(* Logix 5000 project; controller VET 1756-L62 rev 19.52; software revision 19.01; part 8 of 27 *)

        [27].Data.tolva[7] := 17, [27].Data.tolva[8] := 18, [27].Data.tolva[9] := 19, [27].Data.tolva[10] := 20, [27].Data.tolva[11] := 29, [27].Data.tolva[12] := 26, [27].Data.tolva[13] := 27, [27].Data.tolva[14] := 28, [27].Data.tolva[15] := 21, [27].Data.tolva[16] := 38, [27].Data.lugar[0] := 1, [27].Data.lugar[1] := 1, [27].Data.lugar[2] := 1, [27].Data.lugar[3] := 1, [27].Data.lugar[4] := 2, [27].Data.lugar[5] := 2, [27].Data.lugar[6] := 2, [27].Data.lugar[7] := 2, [27].Data.lugar[8] := 3, [27].Data.lugar[9] := 3, [27].Data.lugar[10] := 3, [27].Data.lugar[11] := 4, [27].Data.lugar[12] := 4, [27].Data.lugar[13] := 4, [27].Data.lugar[14] := 4, [27].Data.lugar[15] := 3, [27].Data.lugar[16] := 6, [27].Data.flags[0] := 5, [27].Data.flags[1] := 5, [27].Data.flags[2] := 5, [27].Data.flags[3] := 5, [27].Data.flags[4] := 5, [27].Data.flags[5] := 5, [27].Data.flags[6] := 5, [27].Data.flags[7] := 5, [27].Data.flags[8] := 5, [27].Data.flags[9] := 5, [27].Data.flags[10] := 5, [27].Data.flags[11] := 5, [27].Data.flags[12] := 5, [27].Data.flags[13] := 5, [27].Data.flags[14] := 5, [27].Data.flags[15] := 5, [27].Data.flags[16] := 5, [27].Data.fecha_i[0] := 20140324, [27].Data.fecha_i[1] := 20140324, [27].Data.fecha_i[2] := 20140324, [27].Data.fecha_i[3] := 20140324, [27].Data.fecha_i[4] := 20140324, [27].Data.fecha_i[5] := 20140324, [27].Data.fecha_i[6] := 20140324, [27].Data.fecha_i[7] := 20140324, [27].Data.fecha_i[8] := 20140324, [27].Data.fecha_i[9] := 20140324, [27].Data.fecha_i[10] := 20140324, [27].Data.fecha_i[11] := 20140324, [27].Data.fecha_i[12] := 20140324, [27].Data.fecha_i[13] := 20140324, [27].Data.fecha_i[14] := 20140324, [27].Data.fecha_i[15] := 20140324,
        [27].Data.fecha_i[16] := 20140324, [27].Data.fecha_f[0] := 20140324, [27].Data.fecha_f[1] := 20140324, [27].Data.fecha_f[2] := 20140324, [27].Data.fecha_f[3] := 20140324, [27].Data.fecha_f[4] := 20140324, [27].Data.fecha_f[5] := 20140324, [27].Data.fecha_f[6] := 20140324, [27].Data.fecha_f[7] := 20140324, [27].Data.fecha_f[8] := 20140324, [27].Data.fecha_f[9] := 20140324, [27].Data.fecha_f[10] := 20140324, [27].Data.fecha_f[11] := 20140324, [27].Data.fecha_f[12] := 20140324, [27].Data.fecha_f[13] := 20140324, [27].Data.fecha_f[14] := 20140324, [27].Data.fecha_f[15] := 20140324, [27].Data.fecha_f[16] := 20140324, [27].Data.hora_i[0] := 16373539, [27].Data.hora_i[1] := 16375259, [27].Data.hora_i[2] := 16380789, [27].Data.hora_i[3] := 16381714, [27].Data.hora_i[4] := 16373539, [27].Data.hora_i[5] := 16374674, [27].Data.hora_i[6] := 16375794, [27].Data.hora_i[7] := 16380539, [27].Data.hora_i[8] := 16373539, [27].Data.hora_i[9] := 16383864, [27].Data.hora_i[10] := 16393569, [27].Data.hora_i[11] := 16373539, [27].Data.hora_i[12] := 16381754, [27].Data.hora_i[13] := 16392074, [27].Data.hora_i[14] := 16393769, [27].Data.hora_i[15] := 16401384, [27].Data.hora_i[16] := 16404659, [27].Data.hora_f[0] := 16375239, [27].Data.hora_f[1] := 16380769, [27].Data.hora_f[2] := 16381694, [27].Data.hora_f[3] := 16382799, [27].Data.hora_f[4] := 16374654, [27].Data.hora_f[5] := 16375774, [27].Data.hora_f[6] := 16380519, [27].Data.hora_f[7] := 16381269, [27].Data.hora_f[8] := 16383844, [27].Data.hora_f[9] := 16393549, [27].Data.hora_f[10] := 16401364, [27].Data.hora_f[11] := 16381734, [27].Data.hora_f[12] := 16392054, [27].Data.hora_f[13] := 16393749, [27].Data.hora_f[14] := 16394869, [27].Data.hora_f[15] := 16402879, [27].Data.hora_f[16] := 16412864, [28].Head.folio := 40, [28].Head.orden := -3, [28].Head.formula := 'DUMMY$00$00$00$00$00', [28].Head.correlativo := 20, [28].Head.total_batch := 20, [28].Head.peso_teorico := 1733.0, [28].Data.codigo[0] := 51, [28].Data.codigo[1] := 53,
        [28].Data.codigo[2] := 55, [28].Data.codigo[3] := 57, [28].Data.codigo[4] := 60, [28].Data.codigo[5] := 62, [28].Data.codigo[6] := 64, [28].Data.codigo[7] := 66, [28].Data.codigo[8] := 67, [28].Data.codigo[9] := 68, [28].Data.codigo[10] := 69, [28].Data.codigo[11] := 70, [28].Data.codigo[12] := 74, [28].Data.codigo[13] := 75, [28].Data.codigo[14] := 76, [28].Data.codigo[15] := 77, [28].Data.codigo[16] := 81, [28].Data.peso_f[0] := 400.0, [28].Data.peso_f[1] := 350.0, [28].Data.peso_f[2] := 175.0, [28].Data.peso_f[3] := 225.0, [28].Data.peso_f[4] := 125.0, [28].Data.peso_f[5] := 125.0, [28].Data.peso_f[6] := 65.0, [28].Data.peso_f[7] := 65.0, [28].Data.peso_f[8] := 30.0, [28].Data.peso_f[9] := 25.0, [28].Data.peso_f[10] := 17.5, [28].Data.peso_f[11] := 17.5, [28].Data.peso_f[12] := 30.0, [28].Data.peso_f[13] := 5.0, [28].Data.peso_f[14] := 4.0, [28].Data.peso_f[15] := 4.0, [28].Data.peso_f[16] := 70.0, [28].Data.peso_r[0] := 400.74557, [28].Data.peso_r[1] := 350.39438, [28].Data.peso_r[2] := 175.42383, [28].Data.peso_r[3] := 225.02985, [28].Data.peso_r[4] := 125.35709, [28].Data.peso_r[5] := 125.35757, [28].Data.peso_r[6] := 64.76077, [28].Data.peso_r[7] := 65.17856, [28].Data.peso_r[8] := 29.994562, [28].Data.peso_r[9] := 25.012438, [28].Data.peso_r[10] := 17.509579, [28].Data.peso_r[11] := 17.489931, [28].Data.peso_r[12] := 30.008417, [28].Data.peso_r[13] := 5.02573, [28].Data.peso_r[14] := 3.9976578, [28].Data.peso_r[15] := 4.004547, [28].Data.peso_r[16] := 70.10179, [28].Data.tolva[0] := 2, [28].Data.tolva[1] := 4, [28].Data.tolva[2] := 10, [28].Data.tolva[3] := 12, [28].Data.tolva[4] := 7, [28].Data.tolva[5] := 9, [28].Data.tolva[6] := 15, [28].Data.tolva[7] := 17, [28].Data.tolva[8] := 18, [28].Data.tolva[9] := 19, [28].Data.tolva[10] := 20,
        [28].Data.tolva[11] := 29, [28].Data.tolva[12] := 26, [28].Data.tolva[13] := 27, [28].Data.tolva[14] := 28, [28].Data.tolva[15] := 21, [28].Data.tolva[16] := 38, [28].Data.lugar[0] := 1, [28].Data.lugar[1] := 1, [28].Data.lugar[2] := 1, [28].Data.lugar[3] := 1, [28].Data.lugar[4] := 2, [28].Data.lugar[5] := 2, [28].Data.lugar[6] := 2, [28].Data.lugar[7] := 2, [28].Data.lugar[8] := 3, [28].Data.lugar[9] := 3, [28].Data.lugar[10] := 3, [28].Data.lugar[11] := 4, [28].Data.lugar[12] := 4, [28].Data.lugar[13] := 4, [28].Data.lugar[14] := 4, [28].Data.lugar[15] := 3, [28].Data.lugar[16] := 6, [28].Data.flags[0] := 5, [28].Data.flags[1] := 5, [28].Data.flags[2] := 5, [28].Data.flags[3] := 5, [28].Data.flags[4] := 5, [28].Data.flags[5] := 5, [28].Data.flags[6] := 5, [28].Data.flags[7] := 5, [28].Data.flags[8] := 5, [28].Data.flags[9] := 5, [28].Data.flags[10] := 5, [28].Data.flags[11] := 5, [28].Data.flags[12] := 5, [28].Data.flags[13] := 5, [28].Data.flags[14] := 5, [28].Data.flags[15] := 5, [28].Data.flags[16] := 5, [28].Data.fecha_i[0] := 20140324, [28].Data.fecha_i[1] := 20140324, [28].Data.fecha_i[2] := 20140324, [28].Data.fecha_i[3] := 20140324, [28].Data.fecha_i[4] := 20140324, [28].Data.fecha_i[5] := 20140324, [28].Data.fecha_i[6] := 20140324, [28].Data.fecha_i[7] := 20140324, [28].Data.fecha_i[8] := 20140324, [28].Data.fecha_i[9] := 20140324, [28].Data.fecha_i[10] := 20140324, [28].Data.fecha_i[11] := 20140324, [28].Data.fecha_i[12] := 20140324, [28].Data.fecha_i[13] := 20140324, [28].Data.fecha_i[14] := 20140324, [28].Data.fecha_i[15] := 20140324, [28].Data.fecha_i[16] := 20140324, [28].Data.fecha_f[0] := 20140324, [28].Data.fecha_f[1] := 20140324, [28].Data.fecha_f[2] := 20140324,
        [28].Data.fecha_f[3] := 20140324, [28].Data.fecha_f[4] := 20140324, [28].Data.fecha_f[5] := 20140324, [28].Data.fecha_f[6] := 20140324, [28].Data.fecha_f[7] := 20140324, [28].Data.fecha_f[8] := 20140324, [28].Data.fecha_f[9] := 20140324, [28].Data.fecha_f[10] := 20140324, [28].Data.fecha_f[11] := 20140324, [28].Data.fecha_f[12] := 20140324, [28].Data.fecha_f[13] := 20140324, [28].Data.fecha_f[14] := 20140324, [28].Data.fecha_f[15] := 20140324, [28].Data.fecha_f[16] := 20140324, [28].Data.hora_i[0] := 16404664, [28].Data.hora_i[1] := 16410379, [28].Data.hora_i[2] := 16411914, [28].Data.hora_i[3] := 16412839, [28].Data.hora_i[4] := 16404664, [28].Data.hora_i[5] := 16405794, [28].Data.hora_i[6] := 16410919, [28].Data.hora_i[7] := 16411659, [28].Data.hora_i[8] := 16404664, [28].Data.hora_i[9] := 16414989, [28].Data.hora_i[10] := 16424699, [28].Data.hora_i[11] := 16404664, [28].Data.hora_i[12] := 16412859, [28].Data.hora_i[13] := 16423174, [28].Data.hora_i[14] := 16424899, [28].Data.hora_i[15] := 16432524, [28].Data.hora_i[16] := 16435814, [28].Data.hora_f[0] := 16410359, [28].Data.hora_f[1] := 16411894, [28].Data.hora_f[2] := 16412819, [28].Data.hora_f[3] := 16413919, [28].Data.hora_f[4] := 16405774, [28].Data.hora_f[5] := 16410899, [28].Data.hora_f[6] := 16411639, [28].Data.hora_f[7] := 16412374, [28].Data.hora_f[8] := 16414969, [28].Data.hora_f[9] := 16424679, [28].Data.hora_f[10] := 16432504, [28].Data.hora_f[11] := 16412839, [28].Data.hora_f[12] := 16423154, [28].Data.hora_f[13] := 16424879, [28].Data.hora_f[14] := 16425994, [28].Data.hora_f[15] := 16434029, [28].Data.hora_f[16] := 16444014, [29].Head.folio := 40, [29].Head.orden := -3, [29].Head.formula := 'DUMMY$00$00$00$00$00', [29].Head.correlativo := 20, [29].Head.total_batch := 20, [29].Head.peso_teorico := 1733.0, [29].Data.codigo[0] := 51, [29].Data.codigo[1] := 53, [29].Data.codigo[2] := 55, [29].Data.codigo[3] := 57, [29].Data.codigo[4] := 60, [29].Data.codigo[5] := 62,
        [29].Data.codigo[6] := 64, [29].Data.codigo[7] := 66, [29].Data.codigo[8] := 67, [29].Data.codigo[9] := 68, [29].Data.codigo[10] := 69, [29].Data.codigo[11] := 70, [29].Data.codigo[12] := 74, [29].Data.codigo[13] := 75, [29].Data.codigo[14] := 76, [29].Data.codigo[15] := 77, [29].Data.codigo[16] := 81, [29].Data.peso_f[0] := 400.0, [29].Data.peso_f[1] := 350.0, [29].Data.peso_f[2] := 175.0, [29].Data.peso_f[3] := 225.0, [29].Data.peso_f[4] := 125.0, [29].Data.peso_f[5] := 125.0, [29].Data.peso_f[6] := 65.0, [29].Data.peso_f[7] := 65.0, [29].Data.peso_f[8] := 30.0, [29].Data.peso_f[9] := 25.0, [29].Data.peso_f[10] := 17.5, [29].Data.peso_f[11] := 17.5, [29].Data.peso_f[12] := 30.0, [29].Data.peso_f[13] := 5.0, [29].Data.peso_f[14] := 4.0, [29].Data.peso_f[15] := 4.0, [29].Data.peso_f[16] := 70.0, [29].Data.peso_r[0] := 399.58698, [29].Data.peso_r[1] := 350.3239, [29].Data.peso_r[2] := 175.83856, [29].Data.peso_r[3] := 224.96136, [29].Data.peso_r[4] := 124.67243, [29].Data.peso_r[5] := 125.35696, [29].Data.peso_r[6] := 65.3768, [29].Data.peso_r[7] := 64.766815, [29].Data.peso_r[8] := 29.994562, [29].Data.peso_r[9] := 25.012411, [29].Data.peso_r[10] := 17.509384, [29].Data.peso_r[11] := 17.509584, [29].Data.peso_r[12] := 29.994238, [29].Data.peso_r[13] := 4.9850006, [29].Data.peso_r[14] := 4.00441, [29].Data.peso_r[15] := 4.002121, [29].Data.peso_r[16] := 70.10178, [29].Data.tolva[0] := 2, [29].Data.tolva[1] := 4, [29].Data.tolva[2] := 10, [29].Data.tolva[3] := 12, [29].Data.tolva[4] := 7, [29].Data.tolva[5] := 9, [29].Data.tolva[6] := 15, [29].Data.tolva[7] := 17, [29].Data.tolva[8] := 18, [29].Data.tolva[9] := 19, [29].Data.tolva[10] := 20, [29].Data.tolva[11] := 29, [29].Data.tolva[12] := 26, [29].Data.tolva[13] := 27, [29].Data.tolva[14] := 28,
        [29].Data.tolva[15] := 21, [29].Data.tolva[16] := 38, [29].Data.lugar[0] := 1, [29].Data.lugar[1] := 1, [29].Data.lugar[2] := 1, [29].Data.lugar[3] := 1, [29].Data.lugar[4] := 2, [29].Data.lugar[5] := 2, [29].Data.lugar[6] := 2, [29].Data.lugar[7] := 2, [29].Data.lugar[8] := 3, [29].Data.lugar[9] := 3, [29].Data.lugar[10] := 3, [29].Data.lugar[11] := 4, [29].Data.lugar[12] := 4, [29].Data.lugar[13] := 4, [29].Data.lugar[14] := 4, [29].Data.lugar[15] := 3, [29].Data.lugar[16] := 6, [29].Data.flags[0] := 5, [29].Data.flags[1] := 5, [29].Data.flags[2] := 5, [29].Data.flags[3] := 5, [29].Data.flags[4] := 5, [29].Data.flags[5] := 5, [29].Data.flags[6] := 5, [29].Data.flags[7] := 5, [29].Data.flags[8] := 5, [29].Data.flags[9] := 5, [29].Data.flags[10] := 5, [29].Data.flags[11] := 5, [29].Data.flags[12] := 5, [29].Data.flags[13] := 5, [29].Data.flags[14] := 5, [29].Data.flags[15] := 5, [29].Data.flags[16] := 5, [29].Data.fecha_i[0] := 20140324, [29].Data.fecha_i[1] := 20140324, [29].Data.fecha_i[2] := 20140324, [29].Data.fecha_i[3] := 20140324, [29].Data.fecha_i[4] := 20140324, [29].Data.fecha_i[5] := 20140324, [29].Data.fecha_i[6] := 20140324, [29].Data.fecha_i[7] := 20140324, [29].Data.fecha_i[8] := 20140324, [29].Data.fecha_i[9] := 20140324, [29].Data.fecha_i[10] := 20140324, [29].Data.fecha_i[11] := 20140324, [29].Data.fecha_i[12] := 20140324, [29].Data.fecha_i[13] := 20140324, [29].Data.fecha_i[14] := 20140324, [29].Data.fecha_i[15] := 20140324, [29].Data.fecha_i[16] := 20140324, [29].Data.fecha_f[0] := 20140324, [29].Data.fecha_f[1] := 20140324, [29].Data.fecha_f[2] := 20140324, [29].Data.fecha_f[3] := 20140324, [29].Data.fecha_f[4] := 20140324, [29].Data.fecha_f[5] := 20140324, [29].Data.fecha_f[6] := 20140324,
        [29].Data.fecha_f[7] := 20140324, [29].Data.fecha_f[8] := 20140324, [29].Data.fecha_f[9] := 20140324, [29].Data.fecha_f[10] := 20140324, [29].Data.fecha_f[11] := 20140324, [29].Data.fecha_f[12] := 20140324, [29].Data.fecha_f[13] := 20140324, [29].Data.fecha_f[14] := 20140324, [29].Data.fecha_f[15] := 20140324, [29].Data.fecha_f[16] := 20140324, [29].Data.hora_i[0] := 16435819, [29].Data.hora_i[1] := 16441529, [29].Data.hora_i[2] := 16443059, [29].Data.hora_i[3] := 16443994, [29].Data.hora_i[4] := 16435819, [29].Data.hora_i[5] := 16440949, [29].Data.hora_i[6] := 16442074, [29].Data.hora_i[7] := 16442819, [29].Data.hora_i[8] := 16435819, [29].Data.hora_i[9] := 16450144, [29].Data.hora_i[10] := 16455849, [29].Data.hora_i[11] := 16435819, [29].Data.hora_i[12] := 16444034, [29].Data.hora_i[13] := 16454354, [29].Data.hora_i[14] := 16460049, [29].Data.hora_i[15] := 16463669, [29].Data.hora_i[16] := 16470939, [29].Data.hora_f[0] := 16441509, [29].Data.hora_f[1] := 16443039, [29].Data.hora_f[2] := 16443974, [29].Data.hora_f[3] := 16445079, [29].Data.hora_f[4] := 16440929, [29].Data.hora_f[5] := 16442054, [29].Data.hora_f[6] := 16442799, [29].Data.hora_f[7] := 16443539, [29].Data.hora_f[8] := 16450124, [29].Data.hora_f[9] := 16455829, [29].Data.hora_f[10] := 16463649, [29].Data.hora_f[11] := 16444014, [29].Data.hora_f[12] := 16454334, [29].Data.hora_f[13] := 16460029, [29].Data.hora_f[14] := 16461149, [29].Data.hora_f[15] := 16465159, [29].Data.hora_f[16] := 16475144, [30].Head.folio := 40, [30].Head.orden := -3, [30].Head.formula := 'DUMMY$00$00$00$00$00', [30].Head.correlativo := 20, [30].Head.total_batch := 20, [30].Head.peso_teorico := 1733.0, [30].Data.codigo[0] := 51, [30].Data.codigo[1] := 53, [30].Data.codigo[2] := 55, [30].Data.codigo[3] := 57, [30].Data.codigo[4] := 60, [30].Data.codigo[5] := 62, [30].Data.codigo[6] := 64, [30].Data.codigo[7] := 66, [30].Data.codigo[8] := 67, [30].Data.codigo[9] := 68,
        [30].Data.codigo[10] := 69, [30].Data.codigo[11] := 70, [30].Data.codigo[12] := 74, [30].Data.codigo[13] := 75, [30].Data.codigo[14] := 76, [30].Data.codigo[15] := 77, [30].Data.codigo[16] := 81, [30].Data.peso_f[0] := 400.0, [30].Data.peso_f[1] := 350.0, [30].Data.peso_f[2] := 175.0, [30].Data.peso_f[3] := 225.0, [30].Data.peso_f[4] := 125.0, [30].Data.peso_f[5] := 125.0, [30].Data.peso_f[6] := 65.0, [30].Data.peso_f[7] := 65.0, [30].Data.peso_f[8] := 30.0, [30].Data.peso_f[9] := 25.0, [30].Data.peso_f[10] := 17.5, [30].Data.peso_f[11] := 17.5, [30].Data.peso_f[12] := 30.0, [30].Data.peso_f[13] := 5.0, [30].Data.peso_f[14] := 4.0, [30].Data.peso_f[15] := 4.0, [30].Data.peso_f[16] := 70.0, [30].Data.peso_r[0] := 400.74417, [30].Data.peso_r[1] := 350.39444, [30].Data.peso_r[2] := 175.42377, [30].Data.peso_r[3] := 225.03052, [30].Data.peso_r[4] := 125.3572, [30].Data.peso_r[5] := 125.3581, [30].Data.peso_r[6] := 64.7717, [30].Data.peso_r[7] := 65.17816, [30].Data.peso_r[8] := 30.014194, [30].Data.peso_r[9] := 24.973183, [30].Data.peso_r[10] := 17.489918, [30].Data.peso_r[11] := 17.509579, [30].Data.peso_r[12] := 30.013866, [30].Data.peso_r[13] := 5.0257072, [30].Data.peso_r[14] := 3.9946213, [30].Data.peso_r[15] := 3.984726, [30].Data.peso_r[16] := 70.101776, [30].Data.tolva[0] := 2, [30].Data.tolva[1] := 4, [30].Data.tolva[2] := 10, [30].Data.tolva[3] := 12, [30].Data.tolva[4] := 7, [30].Data.tolva[5] := 9, [30].Data.tolva[6] := 15, [30].Data.tolva[7] := 17, [30].Data.tolva[8] := 18, [30].Data.tolva[9] := 19, [30].Data.tolva[10] := 20, [30].Data.tolva[11] := 29, [30].Data.tolva[12] := 26, [30].Data.tolva[13] := 27, [30].Data.tolva[14] := 28, [30].Data.tolva[15] := 21, [30].Data.tolva[16] := 38, [30].Data.lugar[0] := 1, [30].Data.lugar[1] := 1,
        [30].Data.lugar[2] := 1, [30].Data.lugar[3] := 1, [30].Data.lugar[4] := 2, [30].Data.lugar[5] := 2, [30].Data.lugar[6] := 2, [30].Data.lugar[7] := 2, [30].Data.lugar[8] := 3, [30].Data.lugar[9] := 3, [30].Data.lugar[10] := 3, [30].Data.lugar[11] := 4, [30].Data.lugar[12] := 4, [30].Data.lugar[13] := 4, [30].Data.lugar[14] := 4, [30].Data.lugar[15] := 3, [30].Data.lugar[16] := 6, [30].Data.flags[0] := 5, [30].Data.flags[1] := 5, [30].Data.flags[2] := 5, [30].Data.flags[3] := 5, [30].Data.flags[4] := 5, [30].Data.flags[5] := 5, [30].Data.flags[6] := 5, [30].Data.flags[7] := 5, [30].Data.flags[8] := 5, [30].Data.flags[9] := 5, [30].Data.flags[10] := 5, [30].Data.flags[11] := 5, [30].Data.flags[12] := 5, [30].Data.flags[13] := 5, [30].Data.flags[14] := 5, [30].Data.flags[15] := 5, [30].Data.flags[16] := 5, [30].Data.fecha_i[0] := 20140324, [30].Data.fecha_i[1] := 20140324, [30].Data.fecha_i[2] := 20140324, [30].Data.fecha_i[3] := 20140324, [30].Data.fecha_i[4] := 20140324, [30].Data.fecha_i[5] := 20140324, [30].Data.fecha_i[6] := 20140324, [30].Data.fecha_i[7] := 20140324, [30].Data.fecha_i[8] := 20140324, [30].Data.fecha_i[9] := 20140324, [30].Data.fecha_i[10] := 20140324, [30].Data.fecha_i[11] := 20140324, [30].Data.fecha_i[12] := 20140324, [30].Data.fecha_i[13] := 20140324, [30].Data.fecha_i[14] := 20140324, [30].Data.fecha_i[15] := 20140324, [30].Data.fecha_i[16] := 20140324, [30].Data.fecha_f[0] := 20140324, [30].Data.fecha_f[1] := 20140324, [30].Data.fecha_f[2] := 20140324, [30].Data.fecha_f[3] := 20140324, [30].Data.fecha_f[4] := 20140324, [30].Data.fecha_f[5] := 20140324, [30].Data.fecha_f[6] := 20140324, [30].Data.fecha_f[7] := 20140324, [30].Data.fecha_f[8] := 20140324, [30].Data.fecha_f[9] := 20140324, [30].Data.fecha_f[10] := 20140324,
        [30].Data.fecha_f[11] := 20140324, [30].Data.fecha_f[12] := 20140324, [30].Data.fecha_f[13] := 20140324, [30].Data.fecha_f[14] := 20140324, [30].Data.fecha_f[15] := 20140324, [30].Data.fecha_f[16] := 20140324, [30].Data.hora_i[0] := 16470944, [30].Data.hora_i[1] := 16472659, [30].Data.hora_i[2] := 16474194, [30].Data.hora_i[3] := 16475119, [30].Data.hora_i[4] := 16470944, [30].Data.hora_i[5] := 16472074, [30].Data.hora_i[6] := 16473199, [30].Data.hora_i[7] := 16473939, [30].Data.hora_i[8] := 16470944, [30].Data.hora_i[9] := 16481269, [30].Data.hora_i[10] := 16490969, [30].Data.hora_i[11] := 16470944, [30].Data.hora_i[12] := 16475144, [30].Data.hora_i[13] := 16485474, [30].Data.hora_i[14] := 16491179, [30].Data.hora_i[15] := 16494784, [30].Data.hora_i[16] := 16502049, [30].Data.hora_f[0] := 16472639, [30].Data.hora_f[1] := 16474174, [30].Data.hora_f[2] := 16475099, [30].Data.hora_f[3] := 16480199, [30].Data.hora_f[4] := 16472054, [30].Data.hora_f[5] := 16473179, [30].Data.hora_f[6] := 16473919, [30].Data.hora_f[7] := 16474654, [30].Data.hora_f[8] := 16481249, [30].Data.hora_f[9] := 16490949, [30].Data.hora_f[10] := 16494764, [30].Data.hora_f[11] := 16475124, [30].Data.hora_f[12] := 16485454, [30].Data.hora_f[13] := 16491159, [30].Data.hora_f[14] := 16492274, [30].Data.hora_f[15] := 16500264, [30].Data.hora_f[16] := 16510269, [31].Head.folio := 40, [31].Head.orden := -3, [31].Head.formula := 'DUMMY$00$00$00$00$00', [31].Head.correlativo := 20, [31].Head.total_batch := 20, [31].Head.peso_teorico := 1733.0, [31].Data.codigo[0] := 51, [31].Data.codigo[1] := 53, [31].Data.codigo[2] := 55, [31].Data.codigo[3] := 57, [31].Data.codigo[4] := 60, [31].Data.codigo[5] := 62, [31].Data.codigo[6] := 64, [31].Data.codigo[7] := 66, [31].Data.codigo[8] := 67, [31].Data.codigo[9] := 68, [31].Data.codigo[10] := 69, [31].Data.codigo[11] := 70, [31].Data.codigo[12] := 74, [31].Data.codigo[13] := 75,
        [31].Data.codigo[14] := 76, [31].Data.codigo[15] := 77, [31].Data.codigo[16] := 81, [31].Data.peso_f[0] := 400.0, [31].Data.peso_f[1] := 350.0, [31].Data.peso_f[2] := 175.0, [31].Data.peso_f[3] := 225.0, [31].Data.peso_f[4] := 125.0, [31].Data.peso_f[5] := 125.0, [31].Data.peso_f[6] := 65.0, [31].Data.peso_f[7] := 65.0, [31].Data.peso_f[8] := 30.0, [31].Data.peso_f[9] := 25.0, [31].Data.peso_f[10] := 17.5, [31].Data.peso_f[11] := 17.5, [31].Data.peso_f[12] := 30.0, [31].Data.peso_f[13] := 5.0, [31].Data.peso_f[14] := 4.0, [31].Data.peso_f[15] := 4.0, [31].Data.peso_f[16] := 70.0, [31].Data.peso_r[0] := 399.585, [31].Data.peso_r[1] := 350.3347, [31].Data.peso_r[2] := 174.3056, [31].Data.peso_r[3] := 225.03485, [31].Data.peso_r[4] := 125.35838, [31].Data.peso_r[5] := 124.671875, [31].Data.peso_r[6] := 65.378494, [31].Data.peso_r[7] := 65.382904, [31].Data.peso_r[8] := 29.99456, [31].Data.peso_r[9] := 25.012478, [31].Data.peso_r[10] := 17.506992, [31].Data.peso_r[11] := 17.50707, [31].Data.peso_r[12] := 29.992922, [31].Data.peso_r[13] := 5.0036087, [31].Data.peso_r[14] := 4.004402, [31].Data.peso_r[15] := 4.004532, [31].Data.peso_r[16] := 69.80178, [31].Data.tolva[0] := 2, [31].Data.tolva[1] := 4, [31].Data.tolva[2] := 10, [31].Data.tolva[3] := 12, [31].Data.tolva[4] := 7, [31].Data.tolva[5] := 9, [31].Data.tolva[6] := 15, [31].Data.tolva[7] := 17, [31].Data.tolva[8] := 18, [31].Data.tolva[9] := 19, [31].Data.tolva[10] := 20, [31].Data.tolva[11] := 29, [31].Data.tolva[12] := 26, [31].Data.tolva[13] := 27, [31].Data.tolva[14] := 28, [31].Data.tolva[15] := 21, [31].Data.tolva[16] := 38, [31].Data.lugar[0] := 1, [31].Data.lugar[1] := 1, [31].Data.lugar[2] := 1, [31].Data.lugar[3] := 1, [31].Data.lugar[4] := 2, [31].Data.lugar[5] := 2,
        [31].Data.lugar[6] := 2, [31].Data.lugar[7] := 2, [31].Data.lugar[8] := 3, [31].Data.lugar[9] := 3, [31].Data.lugar[10] := 3, [31].Data.lugar[11] := 4, [31].Data.lugar[12] := 4, [31].Data.lugar[13] := 4, [31].Data.lugar[14] := 4, [31].Data.lugar[15] := 3, [31].Data.lugar[16] := 6, [31].Data.flags[0] := 5, [31].Data.flags[1] := 5, [31].Data.flags[2] := 5, [31].Data.flags[3] := 5, [31].Data.flags[4] := 5, [31].Data.flags[5] := 5, [31].Data.flags[6] := 5, [31].Data.flags[7] := 5, [31].Data.flags[8] := 5, [31].Data.flags[9] := 5, [31].Data.flags[10] := 5, [31].Data.flags[11] := 5, [31].Data.flags[12] := 5, [31].Data.flags[13] := 5, [31].Data.flags[14] := 5, [31].Data.flags[15] := 5, [31].Data.flags[16] := 5, [31].Data.fecha_i[0] := 20140324, [31].Data.fecha_i[1] := 20140324, [31].Data.fecha_i[2] := 20140324, [31].Data.fecha_i[3] := 20140324, [31].Data.fecha_i[4] := 20140324, [31].Data.fecha_i[5] := 20140324, [31].Data.fecha_i[6] := 20140324, [31].Data.fecha_i[7] := 20140324, [31].Data.fecha_i[8] := 20140324, [31].Data.fecha_i[9] := 20140324, [31].Data.fecha_i[10] := 20140324, [31].Data.fecha_i[11] := 20140324, [31].Data.fecha_i[12] := 20140324, [31].Data.fecha_i[13] := 20140324, [31].Data.fecha_i[14] := 20140324, [31].Data.fecha_i[15] := 20140324, [31].Data.fecha_i[16] := 20140324, [31].Data.fecha_f[0] := 20140324, [31].Data.fecha_f[1] := 20140324, [31].Data.fecha_f[2] := 20140324, [31].Data.fecha_f[3] := 20140324, [31].Data.fecha_f[4] := 20140324, [31].Data.fecha_f[5] := 20140324, [31].Data.fecha_f[6] := 20140324, [31].Data.fecha_f[7] := 20140324, [31].Data.fecha_f[8] := 20140324, [31].Data.fecha_f[9] := 20140324, [31].Data.fecha_f[10] := 20140324, [31].Data.fecha_f[11] := 20140324, [31].Data.fecha_f[12] := 20140324, [31].Data.fecha_f[13] := 20140324, [31].Data.fecha_f[14] := 20140324,
        [31].Data.fecha_f[15] := 20140324, [31].Data.fecha_f[16] := 20140324, [31].Data.hora_i[0] := 16502054, [31].Data.hora_i[1] := 16503764, [31].Data.hora_i[2] := 16505304, [31].Data.hora_i[3] := 16510229, [31].Data.hora_i[4] := 16502054, [31].Data.hora_i[5] := 16503184, [31].Data.hora_i[6] := 16504309, [31].Data.hora_i[7] := 16505049, [31].Data.hora_i[8] := 16502054, [31].Data.hora_i[9] := 16512379, [31].Data.hora_i[10] := 16522089, [31].Data.hora_i[11] := 16502054, [31].Data.hora_i[12] := 16510269, [31].Data.hora_i[13] := 16520579, [31].Data.hora_i[14] := 16522284, [31].Data.hora_i[15] := 16525909, [31].Data.hora_i[16] := 16533174, [31].Data.hora_f[0] := 16503744, [31].Data.hora_f[1] := 16505284, [31].Data.hora_f[2] := 16510209, [31].Data.hora_f[3] := 16511309, [31].Data.hora_f[4] := 16503164, [31].Data.hora_f[5] := 16504289, [31].Data.hora_f[6] := 16505029, [31].Data.hora_f[7] := 16505764, [31].Data.hora_f[8] := 16512359, [31].Data.hora_f[9] := 16522069, [31].Data.hora_f[10] := 16525889, [31].Data.hora_f[11] := 16510249, [31].Data.hora_f[12] := 16520559, [31].Data.hora_f[13] := 16522264, [31].Data.hora_f[14] := 16523384, [31].Data.hora_f[15] := 16531389, [31].Data.hora_f[16] := 16541369, [32].Head.folio := 40, [32].Head.orden := -3, [32].Head.formula := 'DUMMY$00$00$00$00$00', [32].Head.correlativo := 20, [32].Head.total_batch := 20, [32].Head.peso_teorico := 1733.0, [32].Data.codigo[0] := 51, [32].Data.codigo[1] := 53, [32].Data.codigo[2] := 55, [32].Data.codigo[3] := 57, [32].Data.codigo[4] := 60, [32].Data.codigo[5] := 62, [32].Data.codigo[6] := 64, [32].Data.codigo[7] := 66, [32].Data.codigo[8] := 67, [32].Data.codigo[9] := 68, [32].Data.codigo[10] := 69, [32].Data.codigo[11] := 70, [32].Data.codigo[12] := 74, [32].Data.codigo[13] := 75, [32].Data.codigo[14] := 76, [32].Data.codigo[15] := 77, [32].Data.codigo[16] := 81, [32].Data.peso_f[0] := 400.0,
        [32].Data.peso_f[1] := 350.0, [32].Data.peso_f[2] := 175.0, [32].Data.peso_f[3] := 225.0, [32].Data.peso_f[4] := 125.0, [32].Data.peso_f[5] := 125.0, [32].Data.peso_f[6] := 65.0, [32].Data.peso_f[7] := 65.0, [32].Data.peso_f[8] := 30.0, [32].Data.peso_f[9] := 25.0, [32].Data.peso_f[10] := 17.5, [32].Data.peso_f[11] := 17.5, [32].Data.peso_f[12] := 30.0, [32].Data.peso_f[13] := 5.0, [32].Data.peso_f[14] := 4.0, [32].Data.peso_f[15] := 4.0, [32].Data.peso_f[16] := 70.0, [32].Data.peso_r[0] := 400.74258, [32].Data.peso_r[1] := 350.04794, [32].Data.peso_r[2] := 175.83911, [32].Data.peso_r[3] := 224.9613, [32].Data.peso_r[4] := 124.67255, [32].Data.peso_r[5] := 125.35698, [32].Data.peso_r[6] := 67.1324, [32].Data.peso_r[7] := 64.767395, [32].Data.peso_r[8] := 30.0142, [32].Data.peso_r[9] := 25.012415, [32].Data.peso_r[10] := 17.509373, [32].Data.peso_r[11] := 17.470303, [32].Data.peso_r[12] := 30.013836, [32].Data.peso_r[13] := 4.9850044, [32].Data.peso_r[14] := 4.0044136, [32].Data.peso_r[15] := 4.0021667, [32].Data.peso_r[16] := 70.10178, [32].Data.tolva[0] := 2, [32].Data.tolva[1] := 4, [32].Data.tolva[2] := 10, [32].Data.tolva[3] := 12, [32].Data.tolva[4] := 7, [32].Data.tolva[5] := 9, [32].Data.tolva[6] := 15, [32].Data.tolva[7] := 17, [32].Data.tolva[8] := 18, [32].Data.tolva[9] := 19, [32].Data.tolva[10] := 20, [32].Data.tolva[11] := 29, [32].Data.tolva[12] := 26, [32].Data.tolva[13] := 27, [32].Data.tolva[14] := 28, [32].Data.tolva[15] := 21, [32].Data.tolva[16] := 38, [32].Data.lugar[0] := 1, [32].Data.lugar[1] := 1, [32].Data.lugar[2] := 1, [32].Data.lugar[3] := 1, [32].Data.lugar[4] := 2, [32].Data.lugar[5] := 2, [32].Data.lugar[6] := 2, [32].Data.lugar[7] := 2, [32].Data.lugar[8] := 3, [32].Data.lugar[9] := 3,
        [32].Data.lugar[10] := 3, [32].Data.lugar[11] := 4, [32].Data.lugar[12] := 4, [32].Data.lugar[13] := 4, [32].Data.lugar[14] := 4, [32].Data.lugar[15] := 3, [32].Data.lugar[16] := 6, [32].Data.flags[0] := 5, [32].Data.flags[1] := 5, [32].Data.flags[2] := 5, [32].Data.flags[3] := 5, [32].Data.flags[4] := 5, [32].Data.flags[5] := 5, [32].Data.flags[6] := 5, [32].Data.flags[7] := 5, [32].Data.flags[8] := 5, [32].Data.flags[9] := 5, [32].Data.flags[10] := 5, [32].Data.flags[11] := 5, [32].Data.flags[12] := 5, [32].Data.flags[13] := 5, [32].Data.flags[14] := 5, [32].Data.flags[15] := 5, [32].Data.flags[16] := 5, [32].Data.fecha_i[0] := 20140324, [32].Data.fecha_i[1] := 20140324, [32].Data.fecha_i[2] := 20140324, [32].Data.fecha_i[3] := 20140324, [32].Data.fecha_i[4] := 20140324, [32].Data.fecha_i[5] := 20140324, [32].Data.fecha_i[6] := 20140324, [32].Data.fecha_i[7] := 20140324, [32].Data.fecha_i[8] := 20140324, [32].Data.fecha_i[9] := 20140324, [32].Data.fecha_i[10] := 20140324, [32].Data.fecha_i[11] := 20140324, [32].Data.fecha_i[12] := 20140324, [32].Data.fecha_i[13] := 20140324, [32].Data.fecha_i[14] := 20140324, [32].Data.fecha_i[15] := 20140324, [32].Data.fecha_i[16] := 20140324, [32].Data.fecha_f[0] := 20140324, [32].Data.fecha_f[1] := 20140324, [32].Data.fecha_f[2] := 20140324, [32].Data.fecha_f[3] := 20140324, [32].Data.fecha_f[4] := 20140324, [32].Data.fecha_f[5] := 20140324, [32].Data.fecha_f[6] := 20140324, [32].Data.fecha_f[7] := 20140324, [32].Data.fecha_f[8] := 20140324, [32].Data.fecha_f[9] := 20140324, [32].Data.fecha_f[10] := 20140324, [32].Data.fecha_f[11] := 20140324, [32].Data.fecha_f[12] := 20140324, [32].Data.fecha_f[13] := 20140324, [32].Data.fecha_f[14] := 20140324, [32].Data.fecha_f[15] := 20140324, [32].Data.fecha_f[16] := 20140324, [32].Data.hora_i[0] := 16533179, [32].Data.hora_i[1] := 16534899,
        [32].Data.hora_i[2] := 16540429, [32].Data.hora_i[3] := 16541354, [32].Data.hora_i[4] := 16533179, [32].Data.hora_i[5] := 16534309, [32].Data.hora_i[6] := 16535434, [32].Data.hora_i[7] := 17425149, [32].Data.hora_i[8] := 16533179, [32].Data.hora_i[9] := 16543504, [32].Data.hora_i[10] := 16553209, [32].Data.hora_i[11] := 16533179, [32].Data.hora_i[12] := 16541389, [32].Data.hora_i[13] := 16551709, [32].Data.hora_i[14] := 16553409, [32].Data.hora_i[15] := 16561024, [32].Data.hora_i[16] := 17431134, [32].Data.hora_f[0] := 16534879, [32].Data.hora_f[1] := 16540409, [32].Data.hora_f[2] := 16541334, [32].Data.hora_f[3] := 16542439, [32].Data.hora_f[4] := 16534289, [32].Data.hora_f[5] := 16535414, [32].Data.hora_f[6] := 17425129, [32].Data.hora_f[7] := 17425869, [32].Data.hora_f[8] := 16543484, [32].Data.hora_f[9] := 16553189, [32].Data.hora_f[10] := 16561004, [32].Data.hora_f[11] := 16541369, [32].Data.hora_f[12] := 16551689, [32].Data.hora_f[13] := 16553389, [32].Data.hora_f[14] := 16554509, [32].Data.hora_f[15] := 16562514, [32].Data.hora_f[16] := 17435334, [33].Head.folio := 40, [33].Head.orden := -3, [33].Head.formula := 'DUMMY$00$00$00$00$00', [33].Head.correlativo := 20, [33].Head.total_batch := 20, [33].Head.peso_teorico := 1733.0, [33].Data.codigo[0] := 51, [33].Data.codigo[1] := 53, [33].Data.codigo[2] := 55, [33].Data.codigo[3] := 57, [33].Data.codigo[4] := 60, [33].Data.codigo[5] := 62, [33].Data.codigo[6] := 64, [33].Data.codigo[7] := 66, [33].Data.codigo[8] := 67, [33].Data.codigo[9] := 68, [33].Data.codigo[10] := 69, [33].Data.codigo[11] := 70, [33].Data.codigo[12] := 74, [33].Data.codigo[13] := 75, [33].Data.codigo[14] := 76, [33].Data.codigo[15] := 77, [33].Data.codigo[16] := 81, [33].Data.peso_f[0] := 400.0, [33].Data.peso_f[1] := 350.0, [33].Data.peso_f[2] := 175.0, [33].Data.peso_f[3] := 225.0, [33].Data.peso_f[4] := 125.0,
        [33].Data.peso_f[5] := 125.0, [33].Data.peso_f[6] := 65.0, [33].Data.peso_f[7] := 65.0, [33].Data.peso_f[8] := 30.0, [33].Data.peso_f[9] := 25.0, [33].Data.peso_f[10] := 17.5, [33].Data.peso_f[11] := 17.5, [33].Data.peso_f[12] := 30.0, [33].Data.peso_f[13] := 5.0, [33].Data.peso_f[14] := 4.0, [33].Data.peso_f[15] := 4.0, [33].Data.peso_f[16] := 70.0, [33].Data.peso_r[0] := 399.58694, [33].Data.peso_r[1] := 350.32443, [33].Data.peso_r[2] := 174.66827, [33].Data.peso_r[3] := 224.96014, [33].Data.peso_r[4] := 124.67244, [33].Data.peso_r[5] := 125.1604, [33].Data.peso_r[6] := 65.37236, [33].Data.peso_r[7] := 65.37787, [33].Data.peso_r[8] := 29.994574, [33].Data.peso_r[9] := 25.012407, [33].Data.peso_r[10] := 17.488525, [33].Data.peso_r[11] := 17.50961, [33].Data.peso_r[12] := 29.99427, [33].Data.peso_r[13] := 5.025669, [33].Data.peso_r[14] := 4.0043983, [33].Data.peso_r[15] := 4.002136, [33].Data.peso_r[16] := 70.10179, [33].Data.tolva[0] := 2, [33].Data.tolva[1] := 4, [33].Data.tolva[2] := 10, [33].Data.tolva[3] := 12, [33].Data.tolva[4] := 7, [33].Data.tolva[5] := 9, [33].Data.tolva[6] := 15, [33].Data.tolva[7] := 17, [33].Data.tolva[8] := 18, [33].Data.tolva[9] := 19, [33].Data.tolva[10] := 20, [33].Data.tolva[11] := 29, [33].Data.tolva[12] := 26, [33].Data.tolva[13] := 27, [33].Data.tolva[14] := 28, [33].Data.tolva[15] := 21, [33].Data.tolva[16] := 38, [33].Data.lugar[0] := 1, [33].Data.lugar[1] := 1, [33].Data.lugar[2] := 1, [33].Data.lugar[3] := 1, [33].Data.lugar[4] := 2, [33].Data.lugar[5] := 2, [33].Data.lugar[6] := 2, [33].Data.lugar[7] := 2, [33].Data.lugar[8] := 3, [33].Data.lugar[9] := 3, [33].Data.lugar[10] := 3, [33].Data.lugar[11] := 4, [33].Data.lugar[12] := 4, [33].Data.lugar[13] := 4,
        [33].Data.lugar[14] := 4, [33].Data.lugar[15] := 3, [33].Data.lugar[16] := 6, [33].Data.flags[0] := 5, [33].Data.flags[1] := 5, [33].Data.flags[2] := 5, [33].Data.flags[3] := 5, [33].Data.flags[4] := 5, [33].Data.flags[5] := 5, [33].Data.flags[6] := 5, [33].Data.flags[7] := 5, [33].Data.flags[8] := 5, [33].Data.flags[9] := 5, [33].Data.flags[10] := 5, [33].Data.flags[11] := 5, [33].Data.flags[12] := 5, [33].Data.flags[13] := 5, [33].Data.flags[14] := 5, [33].Data.flags[15] := 5, [33].Data.flags[16] := 5, [33].Data.fecha_i[0] := 20140324, [33].Data.fecha_i[1] := 20140324, [33].Data.fecha_i[2] := 20140324, [33].Data.fecha_i[3] := 20140324, [33].Data.fecha_i[4] := 20140324, [33].Data.fecha_i[5] := 20140324, [33].Data.fecha_i[6] := 20140324, [33].Data.fecha_i[7] := 20140324, [33].Data.fecha_i[8] := 20140324, [33].Data.fecha_i[9] := 20140324, [33].Data.fecha_i[10] := 20140324, [33].Data.fecha_i[11] := 20140324, [33].Data.fecha_i[12] := 20140324, [33].Data.fecha_i[13] := 20140324, [33].Data.fecha_i[14] := 20140324, [33].Data.fecha_i[15] := 20140324, [33].Data.fecha_i[16] := 20140324, [33].Data.fecha_f[0] := 20140324, [33].Data.fecha_f[1] := 20140324, [33].Data.fecha_f[2] := 20140324, [33].Data.fecha_f[3] := 20140324, [33].Data.fecha_f[4] := 20140324, [33].Data.fecha_f[5] := 20140324, [33].Data.fecha_f[6] := 20140324, [33].Data.fecha_f[7] := 20140324, [33].Data.fecha_f[8] := 20140324, [33].Data.fecha_f[9] := 20140324, [33].Data.fecha_f[10] := 20140324, [33].Data.fecha_f[11] := 20140324, [33].Data.fecha_f[12] := 20140324, [33].Data.fecha_f[13] := 20140324, [33].Data.fecha_f[14] := 20140324, [33].Data.fecha_f[15] := 20140324, [33].Data.fecha_f[16] := 20140324, [33].Data.hora_i[0] := 17431139, [33].Data.hora_i[1] := 17432849, [33].Data.hora_i[2] := 17434379, [33].Data.hora_i[3] := 17435309, [33].Data.hora_i[4] := 17431139, [33].Data.hora_i[5] := 17432274,
        [33].Data.hora_i[6] := 17433394, [33].Data.hora_i[7] := 17434139, [33].Data.hora_i[8] := 17431139, [33].Data.hora_i[9] := 17441464, [33].Data.hora_i[10] := 17451169, [33].Data.hora_i[11] := 17431139, [33].Data.hora_i[12] := 17435354, [33].Data.hora_i[13] := 17445674, [33].Data.hora_i[14] := 17451379, [33].Data.hora_i[15] := 17454984, [33].Data.hora_i[16] := 17462259, [33].Data.hora_f[0] := 17432829, [33].Data.hora_f[1] := 17434359, [33].Data.hora_f[2] := 17435289, [33].Data.hora_f[3] := 17440384, [33].Data.hora_f[4] := 17432254, [33].Data.hora_f[5] := 17433374, [33].Data.hora_f[6] := 17434119, [33].Data.hora_f[7] := 17434864, [33].Data.hora_f[8] := 17441444, [33].Data.hora_f[9] := 17451149, [33].Data.hora_f[10] := 17454964, [33].Data.hora_f[11] := 17435334, [33].Data.hora_f[12] := 17445654, [33].Data.hora_f[13] := 17451359, [33].Data.hora_f[14] := 17452484, [33].Data.hora_f[15] := 17460479, [33].Data.hora_f[16] := 17470464, [34].Head.folio := 38, [34].Head.orden := -3, [34].Head.formula := 'DUMMY$00$00$00$00$00', [34].Head.correlativo := 18, [34].Head.total_batch := 20, [34].Head.peso_teorico := 1733.0, [34].Data.codigo[0] := 51, [34].Data.codigo[1] := 53, [34].Data.codigo[2] := 55, [34].Data.codigo[3] := 57, [34].Data.codigo[4] := 60, [34].Data.codigo[5] := 62, [34].Data.codigo[6] := 64, [34].Data.codigo[7] := 66, [34].Data.codigo[8] := 67, [34].Data.codigo[9] := 68, [34].Data.codigo[10] := 69, [34].Data.codigo[11] := 70, [34].Data.codigo[12] := 74, [34].Data.codigo[13] := 75, [34].Data.codigo[14] := 76, [34].Data.codigo[15] := 77, [34].Data.codigo[16] := 81, [34].Data.peso_f[0] := 400.0, [34].Data.peso_f[1] := 350.0, [34].Data.peso_f[2] := 175.0, [34].Data.peso_f[3] := 225.0, [34].Data.peso_f[4] := 125.0, [34].Data.peso_f[5] := 125.0, [34].Data.peso_f[6] := 65.0, [34].Data.peso_f[7] := 65.0, [34].Data.peso_f[8] := 30.0,
        [34].Data.peso_f[9] := 25.0, [34].Data.peso_f[10] := 17.5, [34].Data.peso_f[11] := 17.5, [34].Data.peso_f[12] := 30.0, [34].Data.peso_f[13] := 5.0, [34].Data.peso_f[14] := 4.0, [34].Data.peso_f[15] := 4.0, [34].Data.peso_f[16] := 70.0, [34].Data.peso_r[0] := 400.74448, [34].Data.peso_r[1] := 350.39426, [34].Data.peso_r[2] := 175.42358, [34].Data.peso_r[3] := 225.02985, [34].Data.peso_r[4] := 125.35715, [34].Data.peso_r[5] := 124.72092, [34].Data.peso_r[6] := 65.37564, [34].Data.peso_r[7] := 65.17847, [34].Data.peso_r[8] := 30.014198, [34].Data.peso_r[9] := 25.012413, [34].Data.peso_r[10] := 17.509575, [34].Data.peso_r[11] := 17.509584, [34].Data.peso_r[12] := 29.99425, [34].Data.peso_r[13] := 5.0060005, [34].Data.peso_r[14] := 4.0019493, [34].Data.peso_r[15] := 4.004524, [34].Data.peso_r[16] := 70.10179, [34].Data.tolva[0] := 2, [34].Data.tolva[1] := 4, [34].Data.tolva[2] := 10, [34].Data.tolva[3] := 12, [34].Data.tolva[4] := 7, [34].Data.tolva[5] := 9, [34].Data.tolva[6] := 15, [34].Data.tolva[7] := 17, [34].Data.tolva[8] := 18, [34].Data.tolva[9] := 19, [34].Data.tolva[10] := 20, [34].Data.tolva[11] := 29, [34].Data.tolva[12] := 26, [34].Data.tolva[13] := 27, [34].Data.tolva[14] := 28, [34].Data.tolva[15] := 21, [34].Data.tolva[16] := 38, [34].Data.lugar[0] := 1, [34].Data.lugar[1] := 1, [34].Data.lugar[2] := 1, [34].Data.lugar[3] := 1, [34].Data.lugar[4] := 2, [34].Data.lugar[5] := 2, [34].Data.lugar[6] := 2, [34].Data.lugar[7] := 2, [34].Data.lugar[8] := 3, [34].Data.lugar[9] := 3, [34].Data.lugar[10] := 3, [34].Data.lugar[11] := 4, [34].Data.lugar[12] := 4, [34].Data.lugar[13] := 4, [34].Data.lugar[14] := 4, [34].Data.lugar[15] := 3, [34].Data.lugar[16] := 6, [34].Data.flags[0] := 5,
        [34].Data.flags[1] := 5, [34].Data.flags[2] := 5, [34].Data.flags[3] := 5, [34].Data.flags[4] := 5, [34].Data.flags[5] := 5, [34].Data.flags[6] := 5, [34].Data.flags[7] := 5, [34].Data.flags[8] := 5, [34].Data.flags[9] := 5, [34].Data.flags[10] := 5, [34].Data.flags[11] := 5, [34].Data.flags[12] := 5, [34].Data.flags[13] := 5, [34].Data.flags[14] := 5, [34].Data.flags[15] := 5, [34].Data.flags[16] := 5, [34].Data.fecha_i[0] := 20140324, [34].Data.fecha_i[1] := 20140324, [34].Data.fecha_i[2] := 20140324, [34].Data.fecha_i[3] := 20140324, [34].Data.fecha_i[4] := 20140324, [34].Data.fecha_i[5] := 20140324, [34].Data.fecha_i[6] := 20140324, [34].Data.fecha_i[7] := 20140324, [34].Data.fecha_i[8] := 20140324, [34].Data.fecha_i[9] := 20140324, [34].Data.fecha_i[10] := 20140324, [34].Data.fecha_i[11] := 20140324, [34].Data.fecha_i[12] := 20140324, [34].Data.fecha_i[13] := 20140324, [34].Data.fecha_i[14] := 20140324, [34].Data.fecha_i[15] := 20140324, [34].Data.fecha_i[16] := 20140324, [34].Data.fecha_f[0] := 20140324, [34].Data.fecha_f[1] := 20140324, [34].Data.fecha_f[2] := 20140324, [34].Data.fecha_f[3] := 20140324, [34].Data.fecha_f[4] := 20140324, [34].Data.fecha_f[5] := 20140324, [34].Data.fecha_f[6] := 20140324, [34].Data.fecha_f[7] := 20140324, [34].Data.fecha_f[8] := 20140324, [34].Data.fecha_f[9] := 20140324, [34].Data.fecha_f[10] := 20140324, [34].Data.fecha_f[11] := 20140324, [34].Data.fecha_f[12] := 20140324, [34].Data.fecha_f[13] := 20140324, [34].Data.fecha_f[14] := 20140324, [34].Data.fecha_f[15] := 20140324, [34].Data.fecha_f[16] := 20140324, [34].Data.hora_i[0] := 17462264, [34].Data.hora_i[1] := 17463979, [34].Data.hora_i[2] := 17465514, [34].Data.hora_i[3] := 17470439, [34].Data.hora_i[4] := 17462264, [34].Data.hora_i[5] := 17463394, [34].Data.hora_i[6] := 17464514, [34].Data.hora_i[7] := 17465259, [34].Data.hora_i[8] := 17462264, [34].Data.hora_i[9] := 17472589,
        [34].Data.hora_i[10] := 17482299, [34].Data.hora_i[11] := 17462264, [34].Data.hora_i[12] := 17470464, [34].Data.hora_i[13] := 17480784, [34].Data.hora_i[14] := 17482494, [34].Data.hora_i[15] := 17490124, [34].Data.hora_i[16] := 17493414, [34].Data.hora_f[0] := 17463959, [34].Data.hora_f[1] := 17465494, [34].Data.hora_f[2] := 17470419, [34].Data.hora_f[3] := 17471519, [34].Data.hora_f[4] := 17463374, [34].Data.hora_f[5] := 17464494, [34].Data.hora_f[6] := 17465239, [34].Data.hora_f[7] := 17465974, [34].Data.hora_f[8] := 17472569, [34].Data.hora_f[9] := 17482279, [34].Data.hora_f[10] := 17490104, [34].Data.hora_f[11] := 17470444, [34].Data.hora_f[12] := 17480764, [34].Data.hora_f[13] := 17482474, [34].Data.hora_f[14] := 17483594, [34].Data.hora_f[15] := 17491629, [34].Data.hora_f[16] := 17501614, [35].Head.folio := 40, [35].Head.orden := -3, [35].Head.formula := 'DUMMY$00$00$00$00$00', [35].Head.correlativo := 20, [35].Head.total_batch := 20, [35].Head.peso_teorico := 1733.0, [35].Data.codigo[0] := 51, [35].Data.codigo[1] := 53, [35].Data.codigo[2] := 55, [35].Data.codigo[3] := 57, [35].Data.codigo[4] := 60, [35].Data.codigo[5] := 62, [35].Data.codigo[6] := 64, [35].Data.codigo[7] := 66, [35].Data.codigo[8] := 67, [35].Data.codigo[9] := 68, [35].Data.codigo[10] := 69, [35].Data.codigo[11] := 70, [35].Data.codigo[12] := 74, [35].Data.codigo[13] := 75, [35].Data.codigo[14] := 76, [35].Data.codigo[15] := 77, [35].Data.codigo[16] := 81, [35].Data.peso_f[0] := 400.0, [35].Data.peso_f[1] := 350.0, [35].Data.peso_f[2] := 175.0, [35].Data.peso_f[3] := 225.0, [35].Data.peso_f[4] := 125.0, [35].Data.peso_f[5] := 125.0, [35].Data.peso_f[6] := 65.0, [35].Data.peso_f[7] := 65.0, [35].Data.peso_f[8] := 30.0, [35].Data.peso_f[9] := 25.0, [35].Data.peso_f[10] := 17.5, [35].Data.peso_f[11] := 17.5, [35].Data.peso_f[12] := 30.0,
        [35].Data.peso_f[13] := 5.0, [35].Data.peso_f[14] := 4.0, [35].Data.peso_f[15] := 4.0, [35].Data.peso_f[16] := 70.0, [35].Data.peso_r[0] := 399.58664, [35].Data.peso_r[1] := 350.32455, [35].Data.peso_r[2] := 174.66797, [35].Data.peso_r[3] := 224.96014, [35].Data.peso_r[4] := 124.67243, [35].Data.peso_r[5] := 125.35694, [35].Data.peso_r[6] := 65.37508, [35].Data.peso_r[7] := 64.76672, [35].Data.peso_r[8] := 29.994583, [35].Data.peso_r[9] := 25.01241, [35].Data.peso_r[10] := 17.50938, [35].Data.peso_r[11] := 17.509592, [35].Data.peso_r[12] := 30.013865, [35].Data.peso_r[13] := 4.9849854, [35].Data.peso_r[14] := 4.0043945, [35].Data.peso_r[15] := 4.002144, [35].Data.peso_r[16] := 70.10179, [35].Data.tolva[0] := 2, [35].Data.tolva[1] := 4, [35].Data.tolva[2] := 10, [35].Data.tolva[3] := 12, [35].Data.tolva[4] := 7, [35].Data.tolva[5] := 9, [35].Data.tolva[6] := 15, [35].Data.tolva[7] := 17, [35].Data.tolva[8] := 18, [35].Data.tolva[9] := 19, [35].Data.tolva[10] := 20, [35].Data.tolva[11] := 29, [35].Data.tolva[12] := 26, [35].Data.tolva[13] := 27, [35].Data.tolva[14] := 28, [35].Data.tolva[15] := 21, [35].Data.tolva[16] := 38, [35].Data.lugar[0] := 1, [35].Data.lugar[1] := 1, [35].Data.lugar[2] := 1, [35].Data.lugar[3] := 1, [35].Data.lugar[4] := 2, [35].Data.lugar[5] := 2, [35].Data.lugar[6] := 2, [35].Data.lugar[7] := 2, [35].Data.lugar[8] := 3, [35].Data.lugar[9] := 3, [35].Data.lugar[10] := 3, [35].Data.lugar[11] := 4, [35].Data.lugar[12] := 4, [35].Data.lugar[13] := 4, [35].Data.lugar[14] := 4, [35].Data.lugar[15] := 3, [35].Data.lugar[16] := 6, [35].Data.flags[0] := 5, [35].Data.flags[1] := 5, [35].Data.flags[2] := 5, [35].Data.flags[3] := 5, [35].Data.flags[4] := 5,
        [35].Data.flags[5] := 5, [35].Data.flags[6] := 5, [35].Data.flags[7] := 5, [35].Data.flags[8] := 5, [35].Data.flags[9] := 5, [35].Data.flags[10] := 5, [35].Data.flags[11] := 5, [35].Data.flags[12] := 5, [35].Data.flags[13] := 5, [35].Data.flags[14] := 5, [35].Data.flags[15] := 5, [35].Data.flags[16] := 5, [35].Data.fecha_i[0] := 20140324, [35].Data.fecha_i[1] := 20140324, [35].Data.fecha_i[2] := 20140324, [35].Data.fecha_i[3] := 20140324, [35].Data.fecha_i[4] := 20140324, [35].Data.fecha_i[5] := 20140324, [35].Data.fecha_i[6] := 20140324, [35].Data.fecha_i[7] := 20140324, [35].Data.fecha_i[8] := 20140324, [35].Data.fecha_i[9] := 20140324, [35].Data.fecha_i[10] := 20140324, [35].Data.fecha_i[11] := 20140324, [35].Data.fecha_i[12] := 20140324, [35].Data.fecha_i[13] := 20140324, [35].Data.fecha_i[14] := 20140324, [35].Data.fecha_i[15] := 20140324, [35].Data.fecha_i[16] := 20140324, [35].Data.fecha_f[0] := 20140324, [35].Data.fecha_f[1] := 20140324, [35].Data.fecha_f[2] := 20140324, [35].Data.fecha_f[3] := 20140324, [35].Data.fecha_f[4] := 20140324, [35].Data.fecha_f[5] := 20140324, [35].Data.fecha_f[6] := 20140324, [35].Data.fecha_f[7] := 20140324, [35].Data.fecha_f[8] := 20140324, [35].Data.fecha_f[9] := 20140324, [35].Data.fecha_f[10] := 20140324, [35].Data.fecha_f[11] := 20140324, [35].Data.fecha_f[12] := 20140324, [35].Data.fecha_f[13] := 20140324, [35].Data.fecha_f[14] := 20140324, [35].Data.fecha_f[15] := 20140324, [35].Data.fecha_f[16] := 20140324, [35].Data.hora_i[0] := 17493419, [35].Data.hora_i[1] := 17495129, [35].Data.hora_i[2] := 17500659, [35].Data.hora_i[3] := 17501589, [35].Data.hora_i[4] := 17493419, [35].Data.hora_i[5] := 17494549, [35].Data.hora_i[6] := 17495674, [35].Data.hora_i[7] := 17500419, [35].Data.hora_i[8] := 17493419, [35].Data.hora_i[9] := 17503744, [35].Data.hora_i[10] := 17513449, [35].Data.hora_i[11] := 17493419, [35].Data.hora_i[12] := 17501634, [35].Data.hora_i[13] := 17511959,
        [35].Data.hora_i[14] := 17513649, [35].Data.hora_i[15] := 17521269, [35].Data.hora_i[16] := 17524539, [35].Data.hora_f[0] := 17495109, [35].Data.hora_f[1] := 17500639, [35].Data.hora_f[2] := 17501569, [35].Data.hora_f[3] := 17502664, [35].Data.hora_f[4] := 17494529, [35].Data.hora_f[5] := 17495654, [35].Data.hora_f[6] := 17500399, [35].Data.hora_f[7] := 17501139, [35].Data.hora_f[8] := 17503724, [35].Data.hora_f[9] := 17513429, [35].Data.hora_f[10] := 17521249, [35].Data.hora_f[11] := 17501614, [35].Data.hora_f[12] := 17511939, [35].Data.hora_f[13] := 17513629, [35].Data.hora_f[14] := 17514749, [35].Data.hora_f[15] := 17522759, [35].Data.hora_f[16] := 17532734, [36].Head.folio := 37, [36].Head.orden := -3, [36].Head.formula := 'DUMMY$00$00$00$00$00', [36].Head.correlativo := 17, [36].Head.total_batch := 20, [36].Head.peso_teorico := 1733.0, [36].Data.codigo[0] := 51, [36].Data.codigo[1] := 53, [36].Data.codigo[2] := 55, [36].Data.codigo[3] := 57, [36].Data.codigo[4] := 60, [36].Data.codigo[5] := 62, [36].Data.codigo[6] := 64, [36].Data.codigo[7] := 66, [36].Data.codigo[8] := 67, [36].Data.codigo[9] := 68, [36].Data.codigo[10] := 69, [36].Data.codigo[11] := 70, [36].Data.codigo[12] := 74, [36].Data.codigo[13] := 75, [36].Data.codigo[14] := 76, [36].Data.codigo[15] := 77, [36].Data.codigo[16] := 81, [36].Data.peso_f[0] := 400.0, [36].Data.peso_f[1] := 350.0, [36].Data.peso_f[2] := 175.0, [36].Data.peso_f[3] := 225.0, [36].Data.peso_f[4] := 125.0, [36].Data.peso_f[5] := 125.0, [36].Data.peso_f[6] := 65.0, [36].Data.peso_f[7] := 65.0, [36].Data.peso_f[8] := 30.0, [36].Data.peso_f[9] := 25.0, [36].Data.peso_f[10] := 17.5, [36].Data.peso_f[11] := 17.5, [36].Data.peso_f[12] := 30.0, [36].Data.peso_f[13] := 5.0, [36].Data.peso_f[14] := 4.0, [36].Data.peso_f[15] := 4.0, [36].Data.peso_f[16] := 70.0,
        [36].Data.peso_r[0] := 400.74445, [36].Data.peso_r[1] := 348.13068, [36].Data.peso_r[2] := 175.77844, [36].Data.peso_r[3] := 225.031, [36].Data.peso_r[4] := 125.357086, [36].Data.peso_r[5] := 125.357956, [36].Data.peso_r[6] := 65.373795, [36].Data.peso_r[7] := 65.17297, [36].Data.peso_r[8] := 29.994598, [36].Data.peso_r[9] := 24.973179, [36].Data.peso_r[10] := 17.489925, [36].Data.peso_r[11] := 17.509586, [36].Data.peso_r[12] := 29.994286, [36].Data.peso_r[13] := 5.0257454, [36].Data.peso_r[14] := 3.9952927, [36].Data.peso_r[15] := 4.004532, [36].Data.peso_r[16] := 70.10178, [36].Data.tolva[0] := 2, [36].Data.tolva[1] := 4, [36].Data.tolva[2] := 10, [36].Data.tolva[3] := 12, [36].Data.tolva[4] := 7, [36].Data.tolva[5] := 9, [36].Data.tolva[6] := 15, [36].Data.tolva[7] := 17, [36].Data.tolva[8] := 18, [36].Data.tolva[9] := 19, [36].Data.tolva[10] := 20, [36].Data.tolva[11] := 29, [36].Data.tolva[12] := 26, [36].Data.tolva[13] := 27, [36].Data.tolva[14] := 28, [36].Data.tolva[15] := 21, [36].Data.tolva[16] := 38, [36].Data.lugar[0] := 1, [36].Data.lugar[1] := 1, [36].Data.lugar[2] := 1, [36].Data.lugar[3] := 1, [36].Data.lugar[4] := 2, [36].Data.lugar[5] := 2, [36].Data.lugar[6] := 2, [36].Data.lugar[7] := 2, [36].Data.lugar[8] := 3, [36].Data.lugar[9] := 3, [36].Data.lugar[10] := 3, [36].Data.lugar[11] := 4, [36].Data.lugar[12] := 4, [36].Data.lugar[13] := 4, [36].Data.lugar[14] := 4, [36].Data.lugar[15] := 3, [36].Data.lugar[16] := 6, [36].Data.flags[0] := 5, [36].Data.flags[1] := 5, [36].Data.flags[2] := 5, [36].Data.flags[3] := 5, [36].Data.flags[4] := 5, [36].Data.flags[5] := 5, [36].Data.flags[6] := 5, [36].Data.flags[7] := 5, [36].Data.flags[8] := 5,
        [36].Data.flags[9] := 5, [36].Data.flags[10] := 5, [36].Data.flags[11] := 5, [36].Data.flags[12] := 5, [36].Data.flags[13] := 5, [36].Data.flags[14] := 5, [36].Data.flags[15] := 5, [36].Data.flags[16] := 5, [36].Data.fecha_i[0] := 20140324, [36].Data.fecha_i[1] := 20140324, [36].Data.fecha_i[2] := 20140324, [36].Data.fecha_i[3] := 20140324, [36].Data.fecha_i[4] := 20140324, [36].Data.fecha_i[5] := 20140324, [36].Data.fecha_i[6] := 20140324, [36].Data.fecha_i[7] := 20140324, [36].Data.fecha_i[8] := 20140324, [36].Data.fecha_i[9] := 20140324, [36].Data.fecha_i[10] := 20140324, [36].Data.fecha_i[11] := 20140324, [36].Data.fecha_i[12] := 20140324, [36].Data.fecha_i[13] := 20140324, [36].Data.fecha_i[14] := 20140324, [36].Data.fecha_i[15] := 20140324, [36].Data.fecha_i[16] := 20140324, [36].Data.fecha_f[0] := 20140324, [36].Data.fecha_f[1] := 20140324, [36].Data.fecha_f[2] := 20140324, [36].Data.fecha_f[3] := 20140324, [36].Data.fecha_f[4] := 20140324, [36].Data.fecha_f[5] := 20140324, [36].Data.fecha_f[6] := 20140324, [36].Data.fecha_f[7] := 20140324, [36].Data.fecha_f[8] := 20140324, [36].Data.fecha_f[9] := 20140324, [36].Data.fecha_f[10] := 20140324, [36].Data.fecha_f[11] := 20140324, [36].Data.fecha_f[12] := 20140324, [36].Data.fecha_f[13] := 20140324, [36].Data.fecha_f[14] := 20140324, [36].Data.fecha_f[15] := 20140324, [36].Data.fecha_f[16] := 20140324, [36].Data.hora_i[0] := 17524544, [36].Data.hora_i[1] := 17530259, [36].Data.hora_i[2] := 17531789, [36].Data.hora_i[3] := 17532719, [36].Data.hora_i[4] := 17524544, [36].Data.hora_i[5] := 17525674, [36].Data.hora_i[6] := 17530799, [36].Data.hora_i[7] := 17531539, [36].Data.hora_i[8] := 17524544, [36].Data.hora_i[9] := 17534869, [36].Data.hora_i[10] := 17544569, [36].Data.hora_i[11] := 17524544, [36].Data.hora_i[12] := 17532744, [36].Data.hora_i[13] := 17543064, [36].Data.hora_i[14] := 17544779, [36].Data.hora_i[15] := 17552384, [36].Data.hora_i[16] := 17555649, [36].Data.hora_f[0] := 17530239,
        [36].Data.hora_f[1] := 17531769, [36].Data.hora_f[2] := 17532699, [36].Data.hora_f[3] := 17533799, [36].Data.hora_f[4] := 17525654, [36].Data.hora_f[5] := 17530779, [36].Data.hora_f[6] := 17531519, [36].Data.hora_f[7] := 17532254, [36].Data.hora_f[8] := 17534849, [36].Data.hora_f[9] := 17544549, [36].Data.hora_f[10] := 17552364, [36].Data.hora_f[11] := 17532724, [36].Data.hora_f[12] := 17543044, [36].Data.hora_f[13] := 17544759, [36].Data.hora_f[14] := 17545874, [36].Data.hora_f[15] := 17553869, [36].Data.hora_f[16] := 17563859, [37].Head.folio := 39, [37].Head.orden := -3, [37].Head.formula := 'DUMMY$00$00$00$00$00', [37].Head.correlativo := 19, [37].Head.total_batch := 20, [37].Head.peso_teorico := 1733.0, [37].Data.codigo[0] := 51, [37].Data.codigo[1] := 53, [37].Data.codigo[2] := 55, [37].Data.codigo[3] := 57, [37].Data.codigo[4] := 60, [37].Data.codigo[5] := 62, [37].Data.codigo[6] := 64, [37].Data.codigo[7] := 66, [37].Data.codigo[8] := 67, [37].Data.codigo[9] := 68, [37].Data.codigo[10] := 69, [37].Data.codigo[11] := 70, [37].Data.codigo[12] := 74, [37].Data.codigo[13] := 75, [37].Data.codigo[14] := 76, [37].Data.codigo[15] := 77, [37].Data.codigo[16] := 81, [37].Data.peso_f[0] := 400.0, [37].Data.peso_f[1] := 350.0, [37].Data.peso_f[2] := 175.0, [37].Data.peso_f[3] := 225.0, [37].Data.peso_f[4] := 125.0, [37].Data.peso_f[5] := 125.0, [37].Data.peso_f[6] := 65.0, [37].Data.peso_f[7] := 65.0, [37].Data.peso_f[8] := 30.0, [37].Data.peso_f[9] := 25.0, [37].Data.peso_f[10] := 17.5, [37].Data.peso_f[11] := 17.5, [37].Data.peso_f[12] := 30.0, [37].Data.peso_f[13] := 5.0, [37].Data.peso_f[14] := 4.0, [37].Data.peso_f[15] := 4.0, [37].Data.peso_f[16] := 70.0, [37].Data.peso_r[0] := 399.58484, [37].Data.peso_r[1] := 350.2168, [37].Data.peso_r[2] := 174.32922, [37].Data.peso_r[3] := 225.03418,
        [37].Data.peso_r[4] := 125.35852, [37].Data.peso_r[5] := 124.672, [37].Data.peso_r[6] := 65.3786, [37].Data.peso_r[7] := 64.771515, [37].Data.peso_r[8] := 30.0142, [37].Data.peso_r[9] := 25.012468, [37].Data.peso_r[10] := 17.506992, [37].Data.peso_r[11] := 17.507055, [37].Data.peso_r[12] := 30.012564, [37].Data.peso_r[13] := 5.003601, [37].Data.peso_r[14] := 4.004406, [37].Data.peso_r[15] := 4.004532, [37].Data.peso_r[16] := 69.801796, [37].Data.tolva[0] := 2, [37].Data.tolva[1] := 4, [37].Data.tolva[2] := 10, [37].Data.tolva[3] := 12, [37].Data.tolva[4] := 7, [37].Data.tolva[5] := 9, [37].Data.tolva[6] := 15, [37].Data.tolva[7] := 17, [37].Data.tolva[8] := 18, [37].Data.tolva[9] := 19, [37].Data.tolva[10] := 20, [37].Data.tolva[11] := 29, [37].Data.tolva[12] := 26, [37].Data.tolva[13] := 27, [37].Data.tolva[14] := 28, [37].Data.tolva[15] := 21, [37].Data.tolva[16] := 38, [37].Data.lugar[0] := 1, [37].Data.lugar[1] := 1, [37].Data.lugar[2] := 1, [37].Data.lugar[3] := 1, [37].Data.lugar[4] := 2, [37].Data.lugar[5] := 2, [37].Data.lugar[6] := 2, [37].Data.lugar[7] := 2, [37].Data.lugar[8] := 3, [37].Data.lugar[9] := 3, [37].Data.lugar[10] := 3, [37].Data.lugar[11] := 4, [37].Data.lugar[12] := 4, [37].Data.lugar[13] := 4, [37].Data.lugar[14] := 4, [37].Data.lugar[15] := 3, [37].Data.lugar[16] := 6, [37].Data.flags[0] := 5, [37].Data.flags[1] := 5, [37].Data.flags[2] := 5, [37].Data.flags[3] := 5, [37].Data.flags[4] := 5, [37].Data.flags[5] := 5, [37].Data.flags[6] := 5, [37].Data.flags[7] := 5, [37].Data.flags[8] := 5, [37].Data.flags[9] := 5, [37].Data.flags[10] := 5, [37].Data.flags[11] := 5, [37].Data.flags[12] := 5,
        [37].Data.flags[13] := 5, [37].Data.flags[14] := 5, [37].Data.flags[15] := 5, [37].Data.flags[16] := 5, [37].Data.fecha_i[0] := 20140324, [37].Data.fecha_i[1] := 20140324, [37].Data.fecha_i[2] := 20140324, [37].Data.fecha_i[3] := 20140324, [37].Data.fecha_i[4] := 20140324, [37].Data.fecha_i[5] := 20140324, [37].Data.fecha_i[6] := 20140324, [37].Data.fecha_i[7] := 20140324, [37].Data.fecha_i[8] := 20140324, [37].Data.fecha_i[9] := 20140324, [37].Data.fecha_i[10] := 20140324, [37].Data.fecha_i[11] := 20140324, [37].Data.fecha_i[12] := 20140324, [37].Data.fecha_i[13] := 20140324, [37].Data.fecha_i[14] := 20140324, [37].Data.fecha_i[15] := 20140324, [37].Data.fecha_i[16] := 20140324, [37].Data.fecha_f[0] := 20140324, [37].Data.fecha_f[1] := 20140324, [37].Data.fecha_f[2] := 20140324, [37].Data.fecha_f[3] := 20140324, [37].Data.fecha_f[4] := 20140324, [37].Data.fecha_f[5] := 20140324, [37].Data.fecha_f[6] := 20140324, [37].Data.fecha_f[7] := 20140324, [37].Data.fecha_f[8] := 20140324, [37].Data.fecha_f[9] := 20140324, [37].Data.fecha_f[10] := 20140324, [37].Data.fecha_f[11] := 20140324, [37].Data.fecha_f[12] := 20140324, [37].Data.fecha_f[13] := 20140324, [37].Data.fecha_f[14] := 20140324, [37].Data.fecha_f[15] := 20140324, [37].Data.fecha_f[16] := 20140324, [37].Data.hora_i[0] := 17555654, [37].Data.hora_i[1] := 17561364, [37].Data.hora_i[2] := 17562904, [37].Data.hora_i[3] := 17563829, [37].Data.hora_i[4] := 17555654, [37].Data.hora_i[5] := 17560784, [37].Data.hora_i[6] := 17561909, [37].Data.hora_i[7] := 17562649, [37].Data.hora_i[8] := 17555654, [37].Data.hora_i[9] := 17565984, [37].Data.hora_i[10] := 17575689, [37].Data.hora_i[11] := 17555654, [37].Data.hora_i[12] := 17563869, [37].Data.hora_i[13] := 17574184, [37].Data.hora_i[14] := 17575889, [37].Data.hora_i[15] := 17583509, [37].Data.hora_i[16] := 17590774, [37].Data.hora_f[0] := 17561344, [37].Data.hora_f[1] := 17562884, [37].Data.hora_f[2] := 17563809, [37].Data.hora_f[3] := 17564909, [37].Data.hora_f[4] := 17560764,
        [37].Data.hora_f[5] := 17561889, [37].Data.hora_f[6] := 17562629, [37].Data.hora_f[7] := 17563359, [37].Data.hora_f[8] := 17565964, [37].Data.hora_f[9] := 17575669, [37].Data.hora_f[10] := 17583489, [37].Data.hora_f[11] := 17563849, [37].Data.hora_f[12] := 17574164, [37].Data.hora_f[13] := 17575869, [37].Data.hora_f[14] := 17580984, [37].Data.hora_f[15] := 17584989, [37].Data.hora_f[16] := 17594969, [38].Head.folio := 30, [38].Head.orden := -3, [38].Head.formula := 'DUMMY$00$00$00$00$00', [38].Head.correlativo := 10, [38].Head.total_batch := 20, [38].Head.peso_teorico := 1733.0, [38].Data.codigo[0] := 51, [38].Data.codigo[1] := 53, [38].Data.codigo[2] := 55, [38].Data.codigo[3] := 57, [38].Data.codigo[4] := 60, [38].Data.codigo[5] := 62, [38].Data.codigo[6] := 64, [38].Data.codigo[7] := 66, [38].Data.codigo[8] := 67, [38].Data.codigo[9] := 68, [38].Data.codigo[10] := 69, [38].Data.codigo[11] := 70, [38].Data.codigo[12] := 74, [38].Data.codigo[13] := 75, [38].Data.codigo[14] := 76, [38].Data.codigo[15] := 77, [38].Data.codigo[16] := 81, [38].Data.peso_f[0] := 400.0, [38].Data.peso_f[1] := 350.0, [38].Data.peso_f[2] := 175.0, [38].Data.peso_f[3] := 225.0, [38].Data.peso_f[4] := 125.0, [38].Data.peso_f[5] := 125.0, [38].Data.peso_f[6] := 65.0, [38].Data.peso_f[7] := 65.0, [38].Data.peso_f[8] := 30.0, [38].Data.peso_f[9] := 25.0, [38].Data.peso_f[10] := 17.5, [38].Data.peso_f[11] := 17.5, [38].Data.peso_f[12] := 30.0, [38].Data.peso_f[13] := 5.0, [38].Data.peso_f[14] := 4.0, [38].Data.peso_f[15] := 4.0, [38].Data.peso_f[16] := 70.0, [38].Data.peso_r[0] := 400.74268, [38].Data.peso_r[1] := 351.1369, [38].Data.peso_r[2] := 174.6651, [38].Data.peso_r[3] := 225.03345, [38].Data.peso_r[4] := 124.672424, [38].Data.peso_r[5] := 125.36279, [38].Data.peso_r[6] := 67.12445, [38].Data.peso_r[7] := 65.37775,
        [38].Data.peso_r[8] := 29.994595, [38].Data.peso_r[9] := 25.01242, [38].Data.peso_r[10] := 17.509396, [38].Data.peso_r[11] := 17.509584, [38].Data.peso_r[12] := 29.994253, [38].Data.peso_r[13] := 4.9851227, [38].Data.peso_r[14] := 4.0043907, [38].Data.peso_r[15] := 4.002121, [38].Data.peso_r[16] := 70.10179, [38].Data.tolva[0] := 2, [38].Data.tolva[1] := 4, [38].Data.tolva[2] := 10, [38].Data.tolva[3] := 12, [38].Data.tolva[4] := 7, [38].Data.tolva[5] := 9, [38].Data.tolva[6] := 15, [38].Data.tolva[7] := 17, [38].Data.tolva[8] := 18, [38].Data.tolva[9] := 19, [38].Data.tolva[10] := 20, [38].Data.tolva[11] := 29, [38].Data.tolva[12] := 26, [38].Data.tolva[13] := 27, [38].Data.tolva[14] := 28, [38].Data.tolva[15] := 21, [38].Data.tolva[16] := 38, [38].Data.lugar[0] := 1, [38].Data.lugar[1] := 1, [38].Data.lugar[2] := 1, [38].Data.lugar[3] := 1, [38].Data.lugar[4] := 2, [38].Data.lugar[5] := 2, [38].Data.lugar[6] := 2, [38].Data.lugar[7] := 2, [38].Data.lugar[8] := 3, [38].Data.lugar[9] := 3, [38].Data.lugar[10] := 3, [38].Data.lugar[11] := 4, [38].Data.lugar[12] := 4, [38].Data.lugar[13] := 4, [38].Data.lugar[14] := 4, [38].Data.lugar[15] := 3, [38].Data.lugar[16] := 6, [38].Data.flags[0] := 5, [38].Data.flags[1] := 5, [38].Data.flags[2] := 5, [38].Data.flags[3] := 5, [38].Data.flags[4] := 5, [38].Data.flags[5] := 5, [38].Data.flags[6] := 5, [38].Data.flags[7] := 5, [38].Data.flags[8] := 5, [38].Data.flags[9] := 5, [38].Data.flags[10] := 5, [38].Data.flags[11] := 5, [38].Data.flags[12] := 5, [38].Data.flags[13] := 5, [38].Data.flags[14] := 5, [38].Data.flags[15] := 5, [38].Data.flags[16] := 5,
        [38].Data.fecha_i[0] := 20140324, [38].Data.fecha_i[1] := 20140324, [38].Data.fecha_i[2] := 20140324, [38].Data.fecha_i[3] := 20140324, [38].Data.fecha_i[4] := 20140324, [38].Data.fecha_i[5] := 20140324, [38].Data.fecha_i[6] := 20140324, [38].Data.fecha_i[7] := 20140324, [38].Data.fecha_i[8] := 20140324, [38].Data.fecha_i[9] := 20140324, [38].Data.fecha_i[10] := 20140324, [38].Data.fecha_i[11] := 20140324, [38].Data.fecha_i[12] := 20140324, [38].Data.fecha_i[13] := 20140324, [38].Data.fecha_i[14] := 20140324, [38].Data.fecha_i[15] := 20140324, [38].Data.fecha_i[16] := 20140324, [38].Data.fecha_f[0] := 20140324, [38].Data.fecha_f[1] := 20140324, [38].Data.fecha_f[2] := 20140324, [38].Data.fecha_f[3] := 20140324, [38].Data.fecha_f[4] := 20140324, [38].Data.fecha_f[5] := 20140324, [38].Data.fecha_f[6] := 20140324, [38].Data.fecha_f[7] := 20140324, [38].Data.fecha_f[8] := 20140324, [38].Data.fecha_f[9] := 20140324, [38].Data.fecha_f[10] := 20140324, [38].Data.fecha_f[11] := 20140324, [38].Data.fecha_f[12] := 20140324, [38].Data.fecha_f[13] := 20140324, [38].Data.fecha_f[14] := 20140324, [38].Data.fecha_f[15] := 20140324, [38].Data.fecha_f[16] := 20140324, [38].Data.hora_i[0] := 18133309, [38].Data.hora_i[1] := 18135019, [38].Data.hora_i[2] := 18140554, [38].Data.hora_i[3] := 18141489, [38].Data.hora_i[4] := 18133309, [38].Data.hora_i[5] := 18134429, [38].Data.hora_i[6] := 18135554, [38].Data.hora_i[7] := 18140969, [38].Data.hora_i[8] := 18133309, [38].Data.hora_i[9] := 18143624, [38].Data.hora_i[10] := 18153329, [38].Data.hora_i[11] := 18133309, [38].Data.hora_i[12] := 18141514, [38].Data.hora_i[13] := 18151834, [38].Data.hora_i[14] := 18153529, [38].Data.hora_i[15] := 18161149, [38].Data.hora_i[16] := 18164419, [38].Data.hora_f[0] := 18134999, [38].Data.hora_f[1] := 18140534, [38].Data.hora_f[2] := 18141469, [38].Data.hora_f[3] := 18142569, [38].Data.hora_f[4] := 18134409, [38].Data.hora_f[5] := 18135534, [38].Data.hora_f[6] := 18140949, [38].Data.hora_f[7] := 18141684, [38].Data.hora_f[8] := 18143604,
        [38].Data.hora_f[9] := 18153309, [38].Data.hora_f[10] := 18161129, [38].Data.hora_f[11] := 18141494, [38].Data.hora_f[12] := 18151814, [38].Data.hora_f[13] := 18153509, [38].Data.hora_f[14] := 18154629, [38].Data.hora_f[15] := 18162639, [38].Data.hora_f[16] := 18172624, [39].Head.folio := 39, [39].Head.orden := -3, [39].Head.formula := 'DUMMY$00$00$00$00$00', [39].Head.correlativo := 19, [39].Head.total_batch := 20, [39].Head.peso_teorico := 1733.0, [39].Data.codigo[0] := 51, [39].Data.codigo[1] := 53, [39].Data.codigo[2] := 55, [39].Data.codigo[3] := 57, [39].Data.codigo[4] := 60, [39].Data.codigo[5] := 62, [39].Data.codigo[6] := 64, [39].Data.codigo[7] := 66, [39].Data.codigo[8] := 67, [39].Data.codigo[9] := 68, [39].Data.codigo[10] := 69, [39].Data.codigo[11] := 70, [39].Data.codigo[12] := 74, [39].Data.codigo[13] := 75, [39].Data.codigo[14] := 76, [39].Data.codigo[15] := 77, [39].Data.codigo[16] := 81, [39].Data.peso_f[0] := 400.0, [39].Data.peso_f[1] := 350.0, [39].Data.peso_f[2] := 175.0, [39].Data.peso_f[3] := 225.0, [39].Data.peso_f[4] := 125.0, [39].Data.peso_f[5] := 125.0, [39].Data.peso_f[6] := 65.0, [39].Data.peso_f[7] := 65.0, [39].Data.peso_f[8] := 30.0, [39].Data.peso_f[9] := 25.0, [39].Data.peso_f[10] := 17.5, [39].Data.peso_f[11] := 17.5, [39].Data.peso_f[12] := 30.0, [39].Data.peso_f[13] := 5.0, [39].Data.peso_f[14] := 4.0, [39].Data.peso_f[15] := 4.0, [39].Data.peso_f[16] := 70.0, [39].Data.peso_r[0] := 399.5864, [39].Data.peso_r[1] := 350.32504, [39].Data.peso_r[2] := 175.83844, [39].Data.peso_r[3] := 224.81665, [39].Data.peso_r[4] := 125.90322, [39].Data.peso_r[5] := 124.67223, [39].Data.peso_r[6] := 65.37846, [39].Data.peso_r[7] := 65.38342, [39].Data.peso_r[8] := 30.014181, [39].Data.peso_r[9] := 25.012465, [39].Data.peso_r[10] := 17.507, [39].Data.peso_r[11] := 17.507072,
        [39].Data.peso_r[12] := 30.012547, [39].Data.peso_r[13] := 5.0035934, [39].Data.peso_r[14] := 4.0043945, [39].Data.peso_r[15] := 4.0045547, [39].Data.peso_r[16] := 70.10179, [39].Data.tolva[0] := 2, [39].Data.tolva[1] := 4, [39].Data.tolva[2] := 10, [39].Data.tolva[3] := 12, [39].Data.tolva[4] := 7, [39].Data.tolva[5] := 9, [39].Data.tolva[6] := 15, [39].Data.tolva[7] := 17, [39].Data.tolva[8] := 18, [39].Data.tolva[9] := 19, [39].Data.tolva[10] := 20, [39].Data.tolva[11] := 29, [39].Data.tolva[12] := 26, [39].Data.tolva[13] := 27, [39].Data.tolva[14] := 28, [39].Data.tolva[15] := 21, [39].Data.tolva[16] := 38, [39].Data.lugar[0] := 1, [39].Data.lugar[1] := 1, [39].Data.lugar[2] := 1, [39].Data.lugar[3] := 1, [39].Data.lugar[4] := 2, [39].Data.lugar[5] := 2, [39].Data.lugar[6] := 2, [39].Data.lugar[7] := 2, [39].Data.lugar[8] := 3, [39].Data.lugar[9] := 3, [39].Data.lugar[10] := 3, [39].Data.lugar[11] := 4, [39].Data.lugar[12] := 4, [39].Data.lugar[13] := 4, [39].Data.lugar[14] := 4, [39].Data.lugar[15] := 3, [39].Data.lugar[16] := 6, [39].Data.flags[0] := 5, [39].Data.flags[1] := 5, [39].Data.flags[2] := 5, [39].Data.flags[3] := 5, [39].Data.flags[4] := 5, [39].Data.flags[5] := 5, [39].Data.flags[6] := 5, [39].Data.flags[7] := 5, [39].Data.flags[8] := 5, [39].Data.flags[9] := 5, [39].Data.flags[10] := 5, [39].Data.flags[11] := 5, [39].Data.flags[12] := 5, [39].Data.flags[13] := 5, [39].Data.flags[14] := 5, [39].Data.flags[15] := 5, [39].Data.flags[16] := 5, [39].Data.fecha_i[0] := 20140324, [39].Data.fecha_i[1] := 20140324, [39].Data.fecha_i[2] := 20140324, [39].Data.fecha_i[3] := 20140324,
        [39].Data.fecha_i[4] := 20140324, [39].Data.fecha_i[5] := 20140324, [39].Data.fecha_i[6] := 20140324, [39].Data.fecha_i[7] := 20140324, [39].Data.fecha_i[8] := 20140324, [39].Data.fecha_i[9] := 20140324, [39].Data.fecha_i[10] := 20140324, [39].Data.fecha_i[11] := 20140324, [39].Data.fecha_i[12] := 20140324, [39].Data.fecha_i[13] := 20140324, [39].Data.fecha_i[14] := 20140324, [39].Data.fecha_i[15] := 20140324, [39].Data.fecha_i[16] := 20140324, [39].Data.fecha_f[0] := 20140324, [39].Data.fecha_f[1] := 20140324, [39].Data.fecha_f[2] := 20140324, [39].Data.fecha_f[3] := 20140324, [39].Data.fecha_f[4] := 20140324, [39].Data.fecha_f[5] := 20140324, [39].Data.fecha_f[6] := 20140324, [39].Data.fecha_f[7] := 20140324, [39].Data.fecha_f[8] := 20140324, [39].Data.fecha_f[9] := 20140324, [39].Data.fecha_f[10] := 20140324, [39].Data.fecha_f[11] := 20140324, [39].Data.fecha_f[12] := 20140324, [39].Data.fecha_f[13] := 20140324, [39].Data.fecha_f[14] := 20140324, [39].Data.fecha_f[15] := 20140324, [39].Data.fecha_f[16] := 20140324, [39].Data.hora_i[0] := 18174929, [39].Data.hora_i[1] := 18180629, [39].Data.hora_i[2] := 18182159, [39].Data.hora_i[3] := 18183099, [39].Data.hora_i[4] := 18174929, [39].Data.hora_i[5] := 18180544, [39].Data.hora_i[6] := 18181669, [39].Data.hora_i[7] := 18182409, [39].Data.hora_i[8] := 18174929, [39].Data.hora_i[9] := 18185249, [39].Data.hora_i[10] := 18194969, [39].Data.hora_i[11] := 18174929, [39].Data.hora_i[12] := 18183149, [39].Data.hora_i[13] := 18193464, [39].Data.hora_i[14] := 18195169, [39].Data.hora_i[15] := 18202789, [39].Data.hora_i[16] := 18210054, [39].Data.hora_f[0] := 18180609, [39].Data.hora_f[1] := 18182139, [39].Data.hora_f[2] := 18183079, [39].Data.hora_f[3] := 18184174, [39].Data.hora_f[4] := 18180524, [39].Data.hora_f[5] := 18181649, [39].Data.hora_f[6] := 18182389, [39].Data.hora_f[7] := 18183124, [39].Data.hora_f[8] := 18185229, [39].Data.hora_f[9] := 18194949, [39].Data.hora_f[10] := 18202769, [39].Data.hora_f[11] := 18183129, [39].Data.hora_f[12] := 18193444,
        [39].Data.hora_f[13] := 18195149, [39].Data.hora_f[14] := 18200264, [39].Data.hora_f[15] := 18204269, [39].Data.hora_f[16] := 18214254, [40].Head.folio := 30, [40].Head.orden := -3, [40].Head.formula := 'DUMMY$00$00$00$00$00', [40].Head.correlativo := 10, [40].Head.total_batch := 20, [40].Head.peso_teorico := 1733.0, [40].Data.codigo[0] := 51, [40].Data.codigo[1] := 53, [40].Data.codigo[2] := 55, [40].Data.codigo[3] := 57, [40].Data.codigo[4] := 60, [40].Data.codigo[5] := 62, [40].Data.codigo[6] := 64, [40].Data.codigo[7] := 66, [40].Data.codigo[8] := 67, [40].Data.codigo[9] := 68, [40].Data.codigo[10] := 69, [40].Data.codigo[11] := 70, [40].Data.codigo[12] := 74, [40].Data.codigo[13] := 75, [40].Data.codigo[14] := 76, [40].Data.codigo[15] := 77, [40].Data.codigo[16] := 81, [40].Data.peso_f[0] := 400.0, [40].Data.peso_f[1] := 350.0, [40].Data.peso_f[2] := 175.0, [40].Data.peso_f[3] := 225.0, [40].Data.peso_f[4] := 125.0, [40].Data.peso_f[5] := 125.0, [40].Data.peso_f[6] := 65.0, [40].Data.peso_f[7] := 65.0, [40].Data.peso_f[8] := 30.0, [40].Data.peso_f[9] := 25.0, [40].Data.peso_f[10] := 17.5, [40].Data.peso_f[11] := 17.5, [40].Data.peso_f[12] := 30.0, [40].Data.peso_f[13] := 5.0, [40].Data.peso_f[14] := 4.0, [40].Data.peso_f[15] := 4.0, [40].Data.peso_f[16] := 70.0, [40].Data.peso_r[0] := 400.7439, [40].Data.peso_r[1] := 350.3952, [40].Data.peso_r[2] := 175.42358, [40].Data.peso_r[3] := 225.02972, [40].Data.peso_r[4] := 125.35715, [40].Data.peso_r[5] := 125.357925, [40].Data.peso_r[6] := 65.32353, [40].Data.peso_r[7] := 65.178406, [40].Data.peso_r[8] := 29.994585, [40].Data.peso_r[9] := 25.01243, [40].Data.peso_r[10] := 17.489902, [40].Data.peso_r[11] := 17.48993, [40].Data.peso_r[12] := 30.008408, [40].Data.peso_r[13] := 5.0257797, [40].Data.peso_r[14] := 3.9952316, [40].Data.peso_r[15] := 3.9847107,
        [40].Data.peso_r[16] := 70.09979, [40].Data.tolva[0] := 2, [40].Data.tolva[1] := 4, [40].Data.tolva[2] := 10, [40].Data.tolva[3] := 12, [40].Data.tolva[4] := 7, [40].Data.tolva[5] := 9, [40].Data.tolva[6] := 15, [40].Data.tolva[7] := 17, [40].Data.tolva[8] := 18, [40].Data.tolva[9] := 19, [40].Data.tolva[10] := 20, [40].Data.tolva[11] := 29, [40].Data.tolva[12] := 26, [40].Data.tolva[13] := 27, [40].Data.tolva[14] := 28, [40].Data.tolva[15] := 21, [40].Data.tolva[16] := 38, [40].Data.lugar[0] := 1, [40].Data.lugar[1] := 1, [40].Data.lugar[2] := 1, [40].Data.lugar[3] := 1, [40].Data.lugar[4] := 2, [40].Data.lugar[5] := 2, [40].Data.lugar[6] := 2, [40].Data.lugar[7] := 2, [40].Data.lugar[8] := 3, [40].Data.lugar[9] := 3, [40].Data.lugar[10] := 3, [40].Data.lugar[11] := 4, [40].Data.lugar[12] := 4, [40].Data.lugar[13] := 4, [40].Data.lugar[14] := 4, [40].Data.lugar[15] := 3, [40].Data.lugar[16] := 6, [40].Data.flags[0] := 5, [40].Data.flags[1] := 5, [40].Data.flags[2] := 5, [40].Data.flags[3] := 5, [40].Data.flags[4] := 5, [40].Data.flags[5] := 5, [40].Data.flags[6] := 5, [40].Data.flags[7] := 5, [40].Data.flags[8] := 5, [40].Data.flags[9] := 5, [40].Data.flags[10] := 5, [40].Data.flags[11] := 5, [40].Data.flags[12] := 5, [40].Data.flags[13] := 5, [40].Data.flags[14] := 5, [40].Data.flags[15] := 5, [40].Data.flags[16] := 5, [40].Data.fecha_i[0] := 20140324, [40].Data.fecha_i[1] := 20140324, [40].Data.fecha_i[2] := 20140324, [40].Data.fecha_i[3] := 20140324, [40].Data.fecha_i[4] := 20140324, [40].Data.fecha_i[5] := 20140324, [40].Data.fecha_i[6] := 20140324, [40].Data.fecha_i[7] := 20140324,
        [40].Data.fecha_i[8] := 20140324, [40].Data.fecha_i[9] := 20140324, [40].Data.fecha_i[10] := 20140324, [40].Data.fecha_i[11] := 20140324, [40].Data.fecha_i[12] := 20140324, [40].Data.fecha_i[13] := 20140324, [40].Data.fecha_i[14] := 20140324, [40].Data.fecha_i[15] := 20140324, [40].Data.fecha_i[16] := 20140324, [40].Data.fecha_f[0] := 20140324, [40].Data.fecha_f[1] := 20140324, [40].Data.fecha_f[2] := 20140324, [40].Data.fecha_f[3] := 20140324, [40].Data.fecha_f[4] := 20140324, [40].Data.fecha_f[5] := 20140324, [40].Data.fecha_f[6] := 20140324, [40].Data.fecha_f[7] := 20140324, [40].Data.fecha_f[8] := 20140324, [40].Data.fecha_f[9] := 20140324, [40].Data.fecha_f[10] := 20140324, [40].Data.fecha_f[11] := 20140324, [40].Data.fecha_f[12] := 20140324, [40].Data.fecha_f[13] := 20140324, [40].Data.fecha_f[14] := 20140324, [40].Data.fecha_f[15] := 20140324, [40].Data.fecha_f[16] := 20140324, [40].Data.hora_i[0] := 18210464, [40].Data.hora_i[1] := 18212179, [40].Data.hora_i[2] := 18213714, [40].Data.hora_i[3] := 18214639, [40].Data.hora_i[4] := 18210464, [40].Data.hora_i[5] := 18211594, [40].Data.hora_i[6] := 18212719, [40].Data.hora_i[7] := 18213459, [40].Data.hora_i[8] := 18210464, [40].Data.hora_i[9] := 18220789, [40].Data.hora_i[10] := 18230499, [40].Data.hora_i[11] := 18210464, [40].Data.hora_i[12] := 18214659, [40].Data.hora_i[13] := 18224974, [40].Data.hora_i[14] := 18230699, [40].Data.hora_i[15] := 18234314, [40].Data.hora_i[16] := 18241569, [40].Data.hora_f[0] := 18212159, [40].Data.hora_f[1] := 18213694, [40].Data.hora_f[2] := 18214619, [40].Data.hora_f[3] := 18215719, [40].Data.hora_f[4] := 18211574, [40].Data.hora_f[5] := 18212699, [40].Data.hora_f[6] := 18213439, [40].Data.hora_f[7] := 18214174, [40].Data.hora_f[8] := 18220769, [40].Data.hora_f[9] := 18230479, [40].Data.hora_f[10] := 18234294, [40].Data.hora_f[11] := 18214639, [40].Data.hora_f[12] := 18224954, [40].Data.hora_f[13] := 18230679, [40].Data.hora_f[14] := 18231794, [40].Data.hora_f[15] := 18235784, [40].Data.hora_f[16] := 18245784,
        [41].Head.folio := 41, [41].Head.orden := -4, [41].Head.formula := 'DUMMY$00$00$00$00$00', [41].Head.correlativo := 1, [41].Head.total_batch := 10, [41].Head.peso_teorico := 1939.6, [41].Data.codigo[0] := 51, [41].Data.codigo[1] := 53, [41].Data.codigo[2] := 55, [41].Data.codigo[3] := 57, [41].Data.codigo[4] := 59, [41].Data.codigo[5] := 60, [41].Data.codigo[6] := 63, [41].Data.codigo[7] := 64, [41].Data.codigo[8] := 67, [41].Data.codigo[9] := 69, [41].Data.codigo[10] := 71, [41].Data.codigo[11] := 73, [41].Data.codigo[12] := 75, [41].Data.codigo[13] := 77, [41].Data.codigo[14] := 79, [41].Data.codigo[15] := 81, [41].Data.codigo[16] := 51, [41].Data.peso_f[0] := 127.85085, [41].Data.peso_f[1] := 320.0, [41].Data.peso_f[2] := 285.0, [41].Data.peso_f[3] := 180.0, [41].Data.peso_f[4] := 160.0, [41].Data.peso_f[5] := 110.0, [41].Data.peso_f[6] := 90.0, [41].Data.peso_f[7] := 90.0, [41].Data.peso_f[8] := 50.0, [41].Data.peso_f[9] := 43.6, [41].Data.peso_f[10] := 35.0, [41].Data.peso_f[11] := 12.0, [41].Data.peso_f[12] := 60.0, [41].Data.peso_f[13] := 56.0, [41].Data.peso_f[14] := 25.0, [41].Data.peso_f[15] := 90.0, [41].Data.peso_f[16] := 205.14914, [41].Data.peso_r[0] := 127.85085, [41].Data.peso_r[1] := 319.9573, [41].Data.peso_r[2] := 284.65698, [41].Data.peso_r[3] := 179.67175, [41].Data.peso_r[4] := 160.38689, [41].Data.peso_r[5] := 110.43254, [41].Data.peso_r[6] := 90.89212, [41].Data.peso_r[7] := 90.33139, [41].Data.peso_r[8] := 49.998474, [41].Data.peso_r[9] := 43.60012, [41].Data.peso_r[10] := 34.952538, [41].Data.peso_r[11] := 11.94725, [41].Data.peso_r[12] := 60.006294, [41].Data.peso_r[13] := 55.99907, [41].Data.peso_r[14] := 24.952972, [41].Data.peso_r[15] := 89.90152, [41].Data.peso_r[16] := 204.69049, [41].Data.tolva[0] := 2, [41].Data.tolva[1] := 4, [41].Data.tolva[2] := 10,
        [41].Data.tolva[3] := 12, [41].Data.tolva[4] := 6, [41].Data.tolva[5] := 7, [41].Data.tolva[6] := 14, [41].Data.tolva[7] := 15, [41].Data.tolva[8] := 18, [41].Data.tolva[9] := 20, [41].Data.tolva[10] := 22, [41].Data.tolva[11] := 24, [41].Data.tolva[12] := 27, [41].Data.tolva[13] := 21, [41].Data.tolva[14] := 31, [41].Data.tolva[15] := 38, [41].Data.tolva[16] := 2, [41].Data.lugar[0] := 1, [41].Data.lugar[1] := 1, [41].Data.lugar[2] := 1, [41].Data.lugar[3] := 1, [41].Data.lugar[4] := 2, [41].Data.lugar[5] := 2, [41].Data.lugar[6] := 2, [41].Data.lugar[7] := 2, [41].Data.lugar[8] := 3, [41].Data.lugar[9] := 3, [41].Data.lugar[10] := 3, [41].Data.lugar[11] := 3, [41].Data.lugar[12] := 4, [41].Data.lugar[13] := 3, [41].Data.lugar[14] := 4, [41].Data.lugar[15] := 6, [41].Data.lugar[16] := 1, [41].Data.flags[0] := 5, [41].Data.flags[1] := 5, [41].Data.flags[2] := 5, [41].Data.flags[3] := 5, [41].Data.flags[4] := 5, [41].Data.flags[5] := 5, [41].Data.flags[6] := 5, [41].Data.flags[7] := 5, [41].Data.flags[8] := 5, [41].Data.flags[9] := 5, [41].Data.flags[10] := 5, [41].Data.flags[11] := 5, [41].Data.flags[12] := 5, [41].Data.flags[13] := 5, [41].Data.flags[14] := 5, [41].Data.flags[15] := 5, [41].Data.flags[16] := 5, [41].Data.fecha_i[0] := 19980101, [41].Data.fecha_i[1] := 19980101, [41].Data.fecha_i[2] := 19980101, [41].Data.fecha_i[3] := 19980101, [41].Data.fecha_i[4] := 19980101, [41].Data.fecha_i[5] := 19980101, [41].Data.fecha_i[6] := 19980101, [41].Data.fecha_i[7] := 19980101, [41].Data.fecha_i[8] := 19980101, [41].Data.fecha_i[9] := 19980101, [41].Data.fecha_i[10] := 19980101, [41].Data.fecha_i[11] := 19980101,
        [41].Data.fecha_i[12] := 19980101, [41].Data.fecha_i[13] := 19980101, [41].Data.fecha_i[14] := 19980101, [41].Data.fecha_i[15] := 19980101, [41].Data.fecha_i[16] := 19980101, [41].Data.fecha_f[0] := 19980101, [41].Data.fecha_f[1] := 19980101, [41].Data.fecha_f[2] := 19980101, [41].Data.fecha_f[3] := 19980101, [41].Data.fecha_f[4] := 19980101, [41].Data.fecha_f[5] := 19980101, [41].Data.fecha_f[6] := 19980101, [41].Data.fecha_f[7] := 19980101, [41].Data.fecha_f[8] := 19980101, [41].Data.fecha_f[9] := 19980101, [41].Data.fecha_f[10] := 19980101, [41].Data.fecha_f[11] := 19980101, [41].Data.fecha_f[12] := 19980101, [41].Data.fecha_f[13] := 19980101, [41].Data.fecha_f[14] := 19980101, [41].Data.fecha_f[15] := 19980101, [41].Data.fecha_f[16] := 19980101, [41].Data.hora_i[0] := 4525013, [41].Data.hora_i[1] := 4541738, [41].Data.hora_i[2] := 4543283, [41].Data.hora_i[3] := 4544693, [41].Data.hora_i[4] := 4525013, [41].Data.hora_i[5] := 4530363, [41].Data.hora_i[6] := 4531393, [41].Data.hora_i[7] := 4533403, [41].Data.hora_i[8] := 4525013, [41].Data.hora_i[9] := 4543328, [41].Data.hora_i[10] := 4560368, [41].Data.hora_i[11] := 4571668, [41].Data.hora_i[12] := 4525013, [41].Data.hora_i[13] := 4574373, [41].Data.hora_i[14] := 4545688, [41].Data.hora_i[15] := 5000473, [41].Data.hora_i[16] := 4545693, [41].Data.hora_f[0] := 4541718, [41].Data.hora_f[1] := 4543263, [41].Data.hora_f[2] := 4544673, [41].Data.hora_f[3] := 4545673, [41].Data.hora_f[4] := 4530343, [41].Data.hora_f[5] := 4531373, [41].Data.hora_f[6] := 4533383, [41].Data.hora_f[7] := 4534288, [41].Data.hora_f[8] := 4543308, [41].Data.hora_f[9] := 4560348, [41].Data.hora_f[10] := 4571648, [41].Data.hora_f[11] := 4574353, [41].Data.hora_f[12] := 4545668, [41].Data.hora_f[13] := 4594268, [41].Data.hora_f[14] := 4555378, [41].Data.hora_f[15] := 5005698, [41].Data.hora_f[16] := 4550768, [42].Head.folio := 42, [42].Head.orden := -4, [42].Head.formula := 'DUMMY$00$00$00$00$00', [42].Head.correlativo := 2,
        [42].Head.total_batch := 10, [42].Head.peso_teorico := 1939.6, [42].Data.codigo[0] := 51, [42].Data.codigo[1] := 53, [42].Data.codigo[2] := 55, [42].Data.codigo[3] := 57, [42].Data.codigo[4] := 59, [42].Data.codigo[5] := 60, [42].Data.codigo[6] := 63, [42].Data.codigo[7] := 64, [42].Data.codigo[8] := 67, [42].Data.codigo[9] := 69, [42].Data.codigo[10] := 71, [42].Data.codigo[11] := 73, [42].Data.codigo[12] := 75, [42].Data.codigo[13] := 77, [42].Data.codigo[14] := 79, [42].Data.codigo[15] := 81, [42].Data.codigo[16] := 51, [42].Data.peso_f[0] := 140.05605, [42].Data.peso_f[1] := 320.0, [42].Data.peso_f[2] := 285.0, [42].Data.peso_f[3] := 180.0, [42].Data.peso_f[4] := 160.0, [42].Data.peso_f[5] := 110.0, [42].Data.peso_f[6] := 90.0, [42].Data.peso_f[7] := 90.0, [42].Data.peso_f[8] := 50.0, [42].Data.peso_f[9] := 43.6, [42].Data.peso_f[10] := 35.0, [42].Data.peso_f[11] := 12.0, [42].Data.peso_f[12] := 60.0, [42].Data.peso_f[13] := 56.0, [42].Data.peso_f[14] := 25.0, [42].Data.peso_f[15] := 90.0, [42].Data.peso_f[16] := 192.94395, [42].Data.peso_r[0] := 140.05605, [42].Data.peso_r[1] := 319.89825, [42].Data.peso_r[2] := 285.71063, [42].Data.peso_r[3] := 179.79224, [42].Data.peso_r[4] := 159.70108, [42].Data.peso_r[5] := 110.48297, [42].Data.peso_r[6] := 90.33145, [42].Data.peso_r[7] := 90.33118, [42].Data.peso_r[8] := 50.00083, [42].Data.peso_r[9] := 43.597755, [42].Data.peso_r[10] := 34.976456, [42].Data.peso_r[11] := 11.966995, [42].Data.peso_r[12] := 60.00628, [42].Data.peso_r[13] := 56.00139, [42].Data.peso_r[14] := 24.9738, [42].Data.peso_r[15] := 90.199486, [42].Data.peso_r[16] := 192.75476, [42].Data.tolva[0] := 2, [42].Data.tolva[1] := 4, [42].Data.tolva[2] := 10, [42].Data.tolva[3] := 12, [42].Data.tolva[4] := 6, [42].Data.tolva[5] := 7, [42].Data.tolva[6] := 14,
        [42].Data.tolva[7] := 15, [42].Data.tolva[8] := 18, [42].Data.tolva[9] := 20, [42].Data.tolva[10] := 22, [42].Data.tolva[11] := 24, [42].Data.tolva[12] := 27, [42].Data.tolva[13] := 21, [42].Data.tolva[14] := 31, [42].Data.tolva[15] := 38, [42].Data.tolva[16] := 3, [42].Data.lugar[0] := 1, [42].Data.lugar[1] := 1, [42].Data.lugar[2] := 1, [42].Data.lugar[3] := 1, [42].Data.lugar[4] := 2, [42].Data.lugar[5] := 2, [42].Data.lugar[6] := 2, [42].Data.lugar[7] := 2, [42].Data.lugar[8] := 3, [42].Data.lugar[9] := 3, [42].Data.lugar[10] := 3, [42].Data.lugar[11] := 3, [42].Data.lugar[12] := 4, [42].Data.lugar[13] := 3, [42].Data.lugar[14] := 4, [42].Data.lugar[15] := 6, [42].Data.lugar[16] := 1, [42].Data.flags[0] := 5, [42].Data.flags[1] := 5, [42].Data.flags[2] := 5, [42].Data.flags[3] := 5, [42].Data.flags[4] := 5, [42].Data.flags[5] := 5, [42].Data.flags[6] := 5, [42].Data.flags[7] := 5, [42].Data.flags[8] := 5, [42].Data.flags[9] := 5, [42].Data.flags[10] := 5, [42].Data.flags[11] := 5, [42].Data.flags[12] := 5, [42].Data.flags[13] := 5, [42].Data.flags[14] := 5, [42].Data.flags[15] := 5, [42].Data.flags[16] := 5, [42].Data.fecha_i[0] := 19980101, [42].Data.fecha_i[1] := 19980101, [42].Data.fecha_i[2] := 19980101, [42].Data.fecha_i[3] := 19980101, [42].Data.fecha_i[4] := 19980101, [42].Data.fecha_i[5] := 19980101, [42].Data.fecha_i[6] := 19980101, [42].Data.fecha_i[7] := 19980101, [42].Data.fecha_i[8] := 19980101, [42].Data.fecha_i[9] := 19980101, [42].Data.fecha_i[10] := 19980101, [42].Data.fecha_i[11] := 19980101, [42].Data.fecha_i[12] := 19980101, [42].Data.fecha_i[13] := 19980101, [42].Data.fecha_i[14] := 19980101, [42].Data.fecha_i[15] := 19980101,
        [42].Data.fecha_i[16] := 19980101, [42].Data.fecha_f[0] := 19980101, [42].Data.fecha_f[1] := 19980101, [42].Data.fecha_f[2] := 19980101, [42].Data.fecha_f[3] := 19980101, [42].Data.fecha_f[4] := 19980101, [42].Data.fecha_f[5] := 19980101, [42].Data.fecha_f[6] := 19980101, [42].Data.fecha_f[7] := 19980101, [42].Data.fecha_f[8] := 19980101, [42].Data.fecha_f[9] := 19980101, [42].Data.fecha_f[10] := 19980101, [42].Data.fecha_f[11] := 19980101, [42].Data.fecha_f[12] := 19980101, [42].Data.fecha_f[13] := 19980101, [42].Data.fecha_f[14] := 19980101, [42].Data.fecha_f[15] := 19980101, [42].Data.fecha_f[16] := 19980101, [42].Data.hora_i[0] := 9150243, [42].Data.hora_i[1] := 9154728, [42].Data.hora_i[2] := 9160708, [42].Data.hora_i[3] := 9162118, [42].Data.hora_i[4] := 9150243, [42].Data.hora_i[5] := 9151593, [42].Data.hora_i[6] := 9152623, [42].Data.hora_i[7] := 9153528, [42].Data.hora_i[8] := 9150243, [42].Data.hora_i[9] := 9164563, [42].Data.hora_i[10] := 9181603, [42].Data.hora_i[11] := 9192923, [42].Data.hora_i[12] := 9150243, [42].Data.hora_i[13] := 9195643, [42].Data.hora_i[14] := 9170963, [42].Data.hora_i[15] := 9221763, [42].Data.hora_i[16] := 9163123, [42].Data.hora_f[0] := 9154708, [42].Data.hora_f[1] := 9160688, [42].Data.hora_f[2] := 9162098, [42].Data.hora_f[3] := 9163103, [42].Data.hora_f[4] := 9151573, [42].Data.hora_f[5] := 9152603, [42].Data.hora_f[6] := 9153508, [42].Data.hora_f[7] := 9154413, [42].Data.hora_f[8] := 9164543, [42].Data.hora_f[9] := 9181583, [42].Data.hora_f[10] := 9192903, [42].Data.hora_f[11] := 9195623, [42].Data.hora_f[12] := 9170943, [42].Data.hora_f[13] := 9215548, [42].Data.hora_f[14] := 9180658, [42].Data.hora_f[15] := 9230978, [42].Data.hora_f[16] := 9164158, [43].Head.folio := 44, [43].Head.orden := -4, [43].Head.formula := 'DUMMY$00$00$00$00$00', [43].Head.correlativo := 4, [43].Head.total_batch := 10, [43].Head.peso_teorico := 1939.6, [43].Data.codigo[0] := 51, [43].Data.codigo[1] := 53,
        [43].Data.codigo[2] := 55, [43].Data.codigo[3] := 57, [43].Data.codigo[4] := 59, [43].Data.codigo[5] := 60, [43].Data.codigo[6] := 63, [43].Data.codigo[7] := 64, [43].Data.codigo[8] := 67, [43].Data.codigo[9] := 69, [43].Data.codigo[10] := 71, [43].Data.codigo[11] := 73, [43].Data.codigo[12] := 75, [43].Data.codigo[13] := 77, [43].Data.codigo[14] := 79, [43].Data.codigo[15] := 81, [43].Data.peso_f[0] := 333.0, [43].Data.peso_f[1] := 320.0, [43].Data.peso_f[2] := 285.0, [43].Data.peso_f[3] := 180.0, [43].Data.peso_f[4] := 160.0, [43].Data.peso_f[5] := 110.0, [43].Data.peso_f[6] := 90.0, [43].Data.peso_f[7] := 90.0, [43].Data.peso_f[8] := 50.0, [43].Data.peso_f[9] := 43.6, [43].Data.peso_f[10] := 35.0, [43].Data.peso_f[11] := 12.0, [43].Data.peso_f[12] := 60.0, [43].Data.peso_f[13] := 56.0, [43].Data.peso_f[14] := 25.0, [43].Data.peso_f[15] := 90.0, [43].Data.peso_r[0] := 333.05017, [43].Data.peso_r[1] := 319.95734, [43].Data.peso_r[2] := 285.7107, [43].Data.peso_r[3] := 179.79156, [43].Data.peso_r[4] := 160.38673, [43].Data.peso_r[5] := 109.831406, [43].Data.peso_r[6] := 90.73453, [43].Data.peso_r[7] := 89.68924, [43].Data.peso_r[8] := 49.999657, [43].Data.peso_r[9] := 43.60013, [43].Data.peso_r[10] := 34.99111, [43].Data.peso_r[11] := 11.985428, [43].Data.peso_r[12] := 25.060871, [43].Data.peso_r[13] := 50.054142, [43].Data.peso_r[14] := 24.992897, [43].Data.peso_r[15] := 90.19949, [43].Data.tolva[0] := 3, [43].Data.tolva[1] := 4, [43].Data.tolva[2] := 10, [43].Data.tolva[3] := 12, [43].Data.tolva[4] := 6, [43].Data.tolva[5] := 7, [43].Data.tolva[6] := 14, [43].Data.tolva[7] := 15, [43].Data.tolva[8] := 18, [43].Data.tolva[9] := 20, [43].Data.tolva[10] := 22, [43].Data.tolva[11] := 24, [43].Data.tolva[12] := 27, [43].Data.tolva[13] := 29,
        [43].Data.tolva[14] := 31, [43].Data.tolva[15] := 38, [43].Data.lugar[0] := 1, [43].Data.lugar[1] := 1, [43].Data.lugar[2] := 1, [43].Data.lugar[3] := 1, [43].Data.lugar[4] := 2, [43].Data.lugar[5] := 2, [43].Data.lugar[6] := 2, [43].Data.lugar[7] := 2, [43].Data.lugar[8] := 3, [43].Data.lugar[9] := 3, [43].Data.lugar[10] := 3, [43].Data.lugar[11] := 3, [43].Data.lugar[12] := 4, [43].Data.lugar[13] := 4, [43].Data.lugar[14] := 4, [43].Data.lugar[15] := 6, [43].Data.flags[0] := 5, [43].Data.flags[1] := 5, [43].Data.flags[2] := 5, [43].Data.flags[3] := 5, [43].Data.flags[4] := 5, [43].Data.flags[5] := 5, [43].Data.flags[6] := 5, [43].Data.flags[7] := 5, [43].Data.flags[8] := 5, [43].Data.flags[9] := 5, [43].Data.flags[10] := 5, [43].Data.flags[11] := 5, [43].Data.flags[12] := 5, [43].Data.flags[13] := 5, [43].Data.flags[14] := 5, [43].Data.flags[15] := 5, [43].Data.fecha_i[0] := 19980101, [43].Data.fecha_i[1] := 19980101, [43].Data.fecha_i[2] := 19980101, [43].Data.fecha_i[3] := 19980101, [43].Data.fecha_i[4] := 19980101, [43].Data.fecha_i[5] := 19980101, [43].Data.fecha_i[6] := 19980101, [43].Data.fecha_i[7] := 19980101, [43].Data.fecha_i[8] := 19980101, [43].Data.fecha_i[9] := 19980101, [43].Data.fecha_i[10] := 19980101, [43].Data.fecha_i[11] := 19980101, [43].Data.fecha_i[12] := 19980101, [43].Data.fecha_i[13] := 19980101, [43].Data.fecha_i[14] := 19980101, [43].Data.fecha_i[15] := 19980101, [43].Data.fecha_f[0] := 19980101, [43].Data.fecha_f[1] := 19980101, [43].Data.fecha_f[2] := 19980101, [43].Data.fecha_f[3] := 19980101, [43].Data.fecha_f[4] := 19980101, [43].Data.fecha_f[5] := 19980101, [43].Data.fecha_f[6] := 19980101, [43].Data.fecha_f[7] := 19980101, [43].Data.fecha_f[8] := 19980101, [43].Data.fecha_f[9] := 19980101,
        [43].Data.fecha_f[10] := 19980101, [43].Data.fecha_f[11] := 19980101, [43].Data.fecha_f[12] := 19980101, [43].Data.fecha_f[13] := 19980101, [43].Data.fecha_f[14] := 19980101, [43].Data.fecha_f[15] := 19980101, [43].Data.hora_i[0] := 9530638, [43].Data.hora_i[1] := 9532223, [43].Data.hora_i[2] := 9533768, [43].Data.hora_i[3] := 9535178, [43].Data.hora_i[4] := 9530638, [43].Data.hora_i[5] := 9531983, [43].Data.hora_i[6] := 9533008, [43].Data.hora_i[7] := 9534423, [43].Data.hora_i[8] := 9530638, [43].Data.hora_i[9] := 9544948, [43].Data.hora_i[10] := 9561988, [43].Data.hora_i[11] := 9573303, [43].Data.hora_i[12] := 9530638, [43].Data.hora_i[13] := 9594453, [43].Data.hora_i[14] := 10023013, [43].Data.hora_i[15] := 10052393, [43].Data.hora_f[0] := 9532203, [43].Data.hora_f[1] := 9533748, [43].Data.hora_f[2] := 9535158, [43].Data.hora_f[3] := 9540163, [43].Data.hora_f[4] := 9531963, [43].Data.hora_f[5] := 9532988, [43].Data.hora_f[6] := 9534403, [43].Data.hora_f[7] := 9535303, [43].Data.hora_f[8] := 9544928, [43].Data.hora_f[9] := 9561968, [43].Data.hora_f[10] := 9573283, [43].Data.hora_f[11] := 9580003, [43].Data.hora_f[12] := 9540523, [43].Data.hora_f[13] := 10022558, [43].Data.hora_f[14] := 10032703, [43].Data.hora_f[15] := 10061623, [44].Head.folio := 45, [44].Head.orden := -4, [44].Head.formula := 'DUMMY$00$00$00$00$00', [44].Head.correlativo := 5, [44].Head.total_batch := 10, [44].Head.peso_teorico := 1939.6, [44].Data.codigo[0] := 51, [44].Data.codigo[1] := 53, [44].Data.codigo[2] := 55, [44].Data.codigo[3] := 57, [44].Data.codigo[4] := 59, [44].Data.codigo[5] := 60, [44].Data.codigo[6] := 63, [44].Data.codigo[7] := 64, [44].Data.codigo[8] := 67, [44].Data.codigo[9] := 69, [44].Data.codigo[10] := 71, [44].Data.codigo[11] := 73, [44].Data.codigo[12] := 75, [44].Data.codigo[13] := 77, [44].Data.codigo[14] := 79, [44].Data.codigo[15] := 81,
        [44].Data.codigo[16] := 75, [44].Data.codigo[17] := 77, [44].Data.peso_f[0] := 333.0, [44].Data.peso_f[1] := 320.0, [44].Data.peso_f[2] := 285.0, [44].Data.peso_f[3] := 180.0, [44].Data.peso_f[4] := 160.0, [44].Data.peso_f[5] := 110.0, [44].Data.peso_f[6] := 90.0, [44].Data.peso_f[7] := 90.0, [44].Data.peso_f[8] := 50.0, [44].Data.peso_f[9] := 43.6, [44].Data.peso_f[10] := 35.0, [44].Data.peso_f[11] := 12.0, [44].Data.peso_f[12] := 50.035057, [44].Data.peso_f[13] := 50.054195, [44].Data.peso_f[14] := 25.0, [44].Data.peso_f[15] := 90.0, [44].Data.peso_f[16] := 9.964943, [44].Data.peso_f[17] := 5.9458046, [44].Data.peso_r[0] := 333.04855, [44].Data.peso_r[1] := 319.95773, [44].Data.peso_r[2] := 285.71063, [44].Data.peso_r[3] := 179.79138, [44].Data.peso_r[4] := 160.3866, [44].Data.peso_r[5] := 109.81894, [44].Data.peso_r[6] := 90.09448, [44].Data.peso_r[7] := 90.330536, [44].Data.peso_r[8] := 49.998447, [44].Data.peso_r[9] := 43.59998, [44].Data.peso_r[10] := 34.991356, [44].Data.peso_r[11] := 12.00528, [44].Data.peso_r[12] := 50.035057, [44].Data.peso_r[13] := 50.054195, [44].Data.peso_r[14] := 24.990486, [44].Data.peso_r[15] := 89.899536, [44].Data.peso_r[16] := 9.976437, [44].Data.peso_r[17] := 5.9526367, [44].Data.tolva[0] := 3, [44].Data.tolva[1] := 4, [44].Data.tolva[2] := 10, [44].Data.tolva[3] := 12, [44].Data.tolva[4] := 6, [44].Data.tolva[5] := 7, [44].Data.tolva[6] := 14, [44].Data.tolva[7] := 15, [44].Data.tolva[8] := 18, [44].Data.tolva[9] := 20, [44].Data.tolva[10] := 22, [44].Data.tolva[11] := 24, [44].Data.tolva[12] := 27, [44].Data.tolva[13] := 29, [44].Data.tolva[14] := 31, [44].Data.tolva[15] := 38, [44].Data.tolva[16] := 27, [44].Data.tolva[17] := 29, [44].Data.lugar[0] := 1, [44].Data.lugar[1] := 1, [44].Data.lugar[2] := 1, [44].Data.lugar[3] := 1,
        [44].Data.lugar[4] := 2, [44].Data.lugar[5] := 2, [44].Data.lugar[6] := 2, [44].Data.lugar[7] := 2, [44].Data.lugar[8] := 3, [44].Data.lugar[9] := 3, [44].Data.lugar[10] := 3, [44].Data.lugar[11] := 3, [44].Data.lugar[12] := 4, [44].Data.lugar[13] := 4, [44].Data.lugar[14] := 4, [44].Data.lugar[15] := 6, [44].Data.lugar[16] := 4, [44].Data.lugar[17] := 4, [44].Data.flags[0] := 5, [44].Data.flags[1] := 5, [44].Data.flags[2] := 5, [44].Data.flags[3] := 5, [44].Data.flags[4] := 5, [44].Data.flags[5] := 5, [44].Data.flags[6] := 5, [44].Data.flags[7] := 5, [44].Data.flags[8] := 5, [44].Data.flags[9] := 5, [44].Data.flags[10] := 5, [44].Data.flags[11] := 5, [44].Data.flags[12] := 5, [44].Data.flags[13] := 5, [44].Data.flags[14] := 5, [44].Data.flags[15] := 5, [44].Data.flags[16] := 5, [44].Data.flags[17] := 5, [44].Data.fecha_i[0] := 19980101, [44].Data.fecha_i[1] := 19980101, [44].Data.fecha_i[2] := 19980101, [44].Data.fecha_i[3] := 19980101, [44].Data.fecha_i[4] := 19980101, [44].Data.fecha_i[5] := 19980101, [44].Data.fecha_i[6] := 19980101, [44].Data.fecha_i[7] := 19980101, [44].Data.fecha_i[8] := 19980101, [44].Data.fecha_i[9] := 19980101, [44].Data.fecha_i[10] := 19980101, [44].Data.fecha_i[11] := 19980101, [44].Data.fecha_i[12] := 19980101, [44].Data.fecha_i[13] := 19980101, [44].Data.fecha_i[14] := 19980101, [44].Data.fecha_i[15] := 19980101, [44].Data.fecha_i[16] := 19980101, [44].Data.fecha_i[17] := 19980101, [44].Data.fecha_f[0] := 19980101, [44].Data.fecha_f[1] := 19980101, [44].Data.fecha_f[2] := 19980101, [44].Data.fecha_f[3] := 19980101, [44].Data.fecha_f[4] := 19980101, [44].Data.fecha_f[5] := 19980101, [44].Data.fecha_f[6] := 19980101, [44].Data.fecha_f[7] := 19980101, [44].Data.fecha_f[8] := 19980101, [44].Data.fecha_f[9] := 19980101,
        [44].Data.fecha_f[10] := 19980101, [44].Data.fecha_f[11] := 19980101, [44].Data.fecha_f[12] := 19980101, [44].Data.fecha_f[13] := 19980101, [44].Data.fecha_f[14] := 19980101, [44].Data.fecha_f[15] := 19980101, [44].Data.fecha_f[16] := 19980101, [44].Data.fecha_f[17] := 19980101, [44].Data.hora_i[0] := 10162287, [44].Data.hora_i[1] := 10163872, [44].Data.hora_i[2] := 10165412, [44].Data.hora_i[3] := 10170827, [44].Data.hora_i[4] := 10162287, [44].Data.hora_i[5] := 10163632, [44].Data.hora_i[6] := 10164657, [44].Data.hora_i[7] := 10165552, [44].Data.hora_i[8] := 10162287, [44].Data.hora_i[9] := 10180602, [44].Data.hora_i[10] := 10193637, [44].Data.hora_i[11] := 10204952, [44].Data.hora_i[12] := 10162287, [44].Data.hora_i[13] := 10181977, [44].Data.hora_i[14] := 10201497, [44].Data.hora_i[15] := 10221612, [44].Data.hora_i[16] := 10211207, [44].Data.hora_i[17] := 10213897, [44].Data.hora_f[0] := 10163852, [44].Data.hora_f[1] := 10165392, [44].Data.hora_f[2] := 10170807, [44].Data.hora_f[3] := 10171817, [44].Data.hora_f[4] := 10163612, [44].Data.hora_f[5] := 10164637, [44].Data.hora_f[6] := 10165532, [44].Data.hora_f[7] := 10170432, [44].Data.hora_f[8] := 10180582, [44].Data.hora_f[9] := 10193617, [44].Data.hora_f[10] := 10204932, [44].Data.hora_f[11] := 10211657, [44].Data.hora_f[12] := 10180917, [44].Data.hora_f[13] := 10201042, [44].Data.hora_f[14] := 10211187, [44].Data.hora_f[15] := 10230822, [44].Data.hora_f[16] := 10213877, [44].Data.hora_f[17] := 10215782, [45].Head.folio := 46, [45].Head.orden := -4, [45].Head.formula := 'DUMMY$00$00$00$00$00', [45].Head.correlativo := 6, [45].Head.total_batch := 10, [45].Head.peso_teorico := 1939.6, [45].Data.codigo[0] := 51, [45].Data.codigo[1] := 53, [45].Data.codigo[2] := 55, [45].Data.codigo[3] := 57, [45].Data.codigo[4] := 59, [45].Data.codigo[5] := 60, [45].Data.codigo[6] := 63, [45].Data.codigo[7] := 64, [45].Data.codigo[8] := 67, [45].Data.codigo[9] := 69,
        [45].Data.codigo[10] := 71, [45].Data.codigo[11] := 73, [45].Data.codigo[12] := 75, [45].Data.codigo[13] := 77, [45].Data.codigo[14] := 79, [45].Data.codigo[15] := 81, [45].Data.peso_f[0] := 333.0, [45].Data.peso_f[1] := 320.0, [45].Data.peso_f[2] := 285.0, [45].Data.peso_f[3] := 180.0, [45].Data.peso_f[4] := 160.0, [45].Data.peso_f[5] := 110.0, [45].Data.peso_f[6] := 90.0, [45].Data.peso_f[7] := 90.0, [45].Data.peso_f[8] := 50.0, [45].Data.peso_f[9] := 43.6, [45].Data.peso_f[10] := 35.0, [45].Data.peso_f[11] := 12.0, [45].Data.peso_f[12] := 60.0, [45].Data.peso_f[13] := 56.0, [45].Data.peso_f[14] := 25.0, [45].Data.peso_f[15] := 90.0, [45].Data.peso_r[0] := 332.91077, [45].Data.peso_r[1] := 319.90942, [45].Data.peso_r[2] := 285.27014, [45].Data.peso_r[3] := 178.66504, [45].Data.peso_r[4] := 159.76216, [45].Data.peso_r[5] := 109.91911, [45].Data.peso_r[6] := 91.76965, [45].Data.peso_r[7] := 90.27219, [45].Data.peso_r[8] := 49.979305, [45].Data.peso_r[9] := 43.60278, [45].Data.peso_r[10] := 34.995293, [45].Data.peso_r[11] := 11.997299, [45].Data.peso_r[12] := 59.986176, [45].Data.peso_r[13] := 56.00318, [45].Data.peso_r[14] := 25.010445, [45].Data.peso_r[15] := 89.91622, [45].Data.tolva[0] := 3, [45].Data.tolva[1] := 4, [45].Data.tolva[2] := 10, [45].Data.tolva[3] := 12, [45].Data.tolva[4] := 6, [45].Data.tolva[5] := 7, [45].Data.tolva[6] := 14, [45].Data.tolva[7] := 15, [45].Data.tolva[8] := 18, [45].Data.tolva[9] := 20, [45].Data.tolva[10] := 22, [45].Data.tolva[11] := 24, [45].Data.tolva[12] := 27, [45].Data.tolva[13] := 29, [45].Data.tolva[14] := 31, [45].Data.tolva[15] := 38, [45].Data.lugar[0] := 1, [45].Data.lugar[1] := 1, [45].Data.lugar[2] := 1, [45].Data.lugar[3] := 1, [45].Data.lugar[4] := 2, [45].Data.lugar[5] := 2,
        [45].Data.lugar[6] := 2, [45].Data.lugar[7] := 2, [45].Data.lugar[8] := 3, [45].Data.lugar[9] := 3, [45].Data.lugar[10] := 3, [45].Data.lugar[11] := 3, [45].Data.lugar[12] := 4, [45].Data.lugar[13] := 4, [45].Data.lugar[14] := 4, [45].Data.lugar[15] := 6, [45].Data.flags[0] := 5, [45].Data.flags[1] := 5, [45].Data.flags[2] := 5, [45].Data.flags[3] := 5, [45].Data.flags[4] := 5, [45].Data.flags[5] := 5, [45].Data.flags[6] := 5, [45].Data.flags[7] := 5, [45].Data.flags[8] := 5, [45].Data.flags[9] := 5, [45].Data.flags[10] := 5, [45].Data.flags[11] := 5, [45].Data.flags[12] := 5, [45].Data.flags[13] := 5, [45].Data.flags[14] := 5, [45].Data.flags[15] := 5, [45].Data.fecha_i[0] := 19980102, [45].Data.fecha_i[1] := 19980102, [45].Data.fecha_i[2] := 19980102, [45].Data.fecha_i[3] := 19980102, [45].Data.fecha_i[4] := 19980102, [45].Data.fecha_i[5] := 19980102, [45].Data.fecha_i[6] := 19980102, [45].Data.fecha_i[7] := 19980102, [45].Data.fecha_i[8] := 19980102, [45].Data.fecha_i[9] := 19980102, [45].Data.fecha_i[10] := 19980102, [45].Data.fecha_i[11] := 19980102, [45].Data.fecha_i[12] := 19980102, [45].Data.fecha_i[13] := 19980102, [45].Data.fecha_i[14] := 19980102, [45].Data.fecha_i[15] := 19980102, [45].Data.fecha_f[0] := 19980102, [45].Data.fecha_f[1] := 19980102, [45].Data.fecha_f[2] := 19980102, [45].Data.fecha_f[3] := 19980102, [45].Data.fecha_f[4] := 19980102, [45].Data.fecha_f[5] := 19980102, [45].Data.fecha_f[6] := 19980102, [45].Data.fecha_f[7] := 19980102, [45].Data.fecha_f[8] := 19980102, [45].Data.fecha_f[9] := 19980102, [45].Data.fecha_f[10] := 19980102, [45].Data.fecha_f[11] := 19980102, [45].Data.fecha_f[12] := 19980102, [45].Data.fecha_f[13] := 19980102, [45].Data.fecha_f[14] := 19980102, [45].Data.fecha_f[15] := 19980102, [45].Data.hora_i[0] := 22322011, [45].Data.hora_i[1] := 22323596,
        [45].Data.hora_i[2] := 22325131, [45].Data.hora_i[3] := 22330536, [45].Data.hora_i[4] := 22384696, [45].Data.hora_i[5] := 22390426, [45].Data.hora_i[6] := 22391451, [45].Data.hora_i[7] := 22393256, [45].Data.hora_i[8] := 22322011, [45].Data.hora_i[9] := 22340321, [45].Data.hora_i[10] := 22353356, [45].Data.hora_i[11] := 22364666, [45].Data.hora_i[12] := 22322011, [45].Data.hora_i[13] := 22342706, [45].Data.hora_i[14] := 22362581, [45].Data.hora_i[15] := 22395501, [45].Data.hora_f[0] := 22323576, [45].Data.hora_f[1] := 22325111, [45].Data.hora_f[2] := 22330516, [45].Data.hora_f[3] := 22331516, [45].Data.hora_f[4] := 22390406, [45].Data.hora_f[5] := 22391431, [45].Data.hora_f[6] := 22393236, [45].Data.hora_f[7] := 22394131, [45].Data.hora_f[8] := 22340301, [45].Data.hora_f[9] := 22353336, [45].Data.hora_f[10] := 22364646, [45].Data.hora_f[11] := 22371361, [45].Data.hora_f[12] := 22342686, [45].Data.hora_f[13] := 22362561, [45].Data.hora_f[14] := 22372251, [45].Data.hora_f[15] := 22404716, [46].Head.folio := 47, [46].Head.orden := -4, [46].Head.formula := 'DUMMY$00$00$00$00$00', [46].Head.correlativo := 7, [46].Head.total_batch := 10, [46].Head.peso_teorico := 1939.6, [46].Data.codigo[0] := 51, [46].Data.codigo[1] := 53, [46].Data.codigo[2] := 55, [46].Data.codigo[3] := 57, [46].Data.codigo[4] := 59, [46].Data.codigo[5] := 60, [46].Data.codigo[6] := 63, [46].Data.codigo[7] := 64, [46].Data.codigo[8] := 67, [46].Data.codigo[9] := 69, [46].Data.codigo[10] := 71, [46].Data.codigo[11] := 73, [46].Data.codigo[12] := 75, [46].Data.codigo[13] := 77, [46].Data.codigo[14] := 79, [46].Data.codigo[15] := 81, [46].Data.peso_f[0] := 333.0, [46].Data.peso_f[1] := 320.0, [46].Data.peso_f[2] := 285.0, [46].Data.peso_f[3] := 180.0, [46].Data.peso_f[4] := 160.0, [46].Data.peso_f[5] := 110.0, [46].Data.peso_f[6] := 90.0, [46].Data.peso_f[7] := 90.0,
